		//ALARMS
	(*Input set1 L1*) 	AddError[w_Index](
			b_ErrorTrig			:= Get.Events.Input[i][phases.L1].b_alarm,
			out_ST_Error			:= a_ActiveEvents[w_Index],
			w_ErrorID					:= ((i -1) * 8) + 5,
			s_Message				:= ConcatMultiString(s1:= 'alarm: input ',
										s2:= TO_STRING(i),
			 							s3:= ' - L1: ',
										s4:= LREAL_TO_FMTSTR(Get.Events.Input[i][phases.L1].r_MaxCurrentDetected,1, TRUE),
										s5:= ' A for ',
										s6:= TO_STRING(Get.Events.Input[i][phases.L1].t_MaxTimeActive)),
			e_sev					:= eseverity.Warning,
			e_ErrAckAccess		:= eErrAckAccess.operator
			);
		w_Index := w_Index +1;
	(*Input set1 L2*) 	AddError[w_Index](
			b_ErrorTrig			:= Get.Events.Input[i][phases.L2].b_alarm,
			out_ST_Error			:= a_ActiveEvents[w_Index],
			w_ErrorID					:= ((i -1) * 8) + 6,
			s_Message				:= ConcatMultiString(s1:= 'alarm: input ',
										s2:= TO_STRING(i),
			 							s3:= ' - L2: ',
										s4:= LREAL_TO_FMTSTR(Get.Events.Input[i][phases.L2].r_MaxCurrentDetected,1, TRUE),
										s5:= ' A for ',
										s6:= TO_STRING(Get.Events.Input[i][phases.L2].t_MaxTimeActive)),
			e_sev					:= eseverity.Warning,
			e_ErrAckAccess		:= eErrAckAccess.operator
			);
		w_Index := w_Index +1;
	(*Input set1 L3*) 	AddError[w_Index](
			b_ErrorTrig			:= Get.Events.Input[i][phases.L3].b_alarm,
			out_ST_Error			:= a_ActiveEvents[w_Index],
			w_ErrorID					:= ((i -1) * 8) + 7,
			s_Message				:= ConcatMultiString(s1:= 'alarm: input ',
										s2:= TO_STRING(i),
			 							s3:= ' - L3: ',
										s4:= LREAL_TO_FMTSTR(Get.Events.Input[i][phases.L3].r_MaxCurrentDetected,1, TRUE),
										s5:= ' A for ',
										s6:= TO_STRING(Get.Events.Input[i][phases.L3].t_MaxTimeActive)),
			e_sev					:= eseverity.Warning,
			e_ErrAckAccess		:= eErrAckAccess.operator
			);
		w_Index := w_Index +1;
	(*Input set1 N*) 	AddError[w_Index](
			b_ErrorTrig			:= Get.Events.Input[i][phases.N].b_alarm,
			out_ST_Error			:= a_ActiveEvents[w_Index],
			w_ErrorID					:= ((i -1) * 8) + 8,
			s_Message				:= ConcatMultiString(s1:= 'alarm: input ',
										s2:= TO_STRING(i),
			 							s3:= ' - N: ',
										s4:= LREAL_TO_FMTSTR(Get.Events.Input[i][phases.N].r_MaxCurrentDetected,1, TRUE),
										s5:= ' A for ',
										s6:= TO_STRING(Get.Events.Input[i][phases.N].t_MaxTimeActive)),
			e_sev					:= eseverity.Warning,
			e_ErrAckAccess		:= eErrAckAccess.operator
			);
		w_Index := w_Index +1;
END_FOR

//OUTPUTS
FOR i:= 1 TO 3 DO
	//Warnings
	(*Input set1 L1*) 	AddError[w_Index](
			b_ErrorTrig			:= Get.Events.Output[i][phases.L1].b_warning,
			out_ST_Error			:= a_ActiveEvents[w_Index],
			w_ErrorID					:= ((i -1) * 8) + 17,
			s_Message				:= ConcatMultiString(s1:= 'warning: output ',
										s2:= TO_STRING(i),
			 							s3:= ' - L1: ',
										s4:= TO_STRING(Get.Events.Output[i][phases.L1].ui_actLoad),
										s5:= ' %, remaining time ',
										s6:= TO_STRING(Get.Events.Output[i][phases.L1].t_RemainingTime)),
			e_sev					:= eseverity.Warning,
			e_ErrAckAccess		:= eErrAckAccess.operator,
			b_autoClear			:= TRUE
			);
		w_Index := w_Index +1;
	(*Input set1 L2*) 	AddError[w_Index](
			b_ErrorTrig			:= Get.Events.Output[i][phases.L2].b_warning,
			out_ST_Error			:= a_ActiveEvents[w_Index],
			w_ErrorID					:= ((i -1) * 8) + 18,
			s_Message				:= ConcatMultiString(s1:= 'warning: output ',
										s2:= TO_STRING(i),
			 							s3:= ' - L2: ',
										s4:= TO_STRING(Get.Events.Output[i][phases.L2].ui_actLoad),
										s5:= ' %, remaining time ',
										s6:= TO_STRING(Get.Events.Output[i][phases.L2].t_RemainingTime)),
			e_sev					:= eseverity.Warning,
			e_ErrAckAccess		:= eErrAckAccess.operator,
			b_autoClear			:= TRUE
			);
		w_Index := w_Index +1;
	(*Input set1 L3*) 	AddError[w_Index](
			b_ErrorTrig			:= Get.Events.Output[i][phases.L3].b_warning,
			out_ST_Error			:= a_ActiveEvents[w_Index],
			w_ErrorID					:= ((i -1) * 8) + 19,
			s_Message				:= ConcatMultiString(s1:= 'warning: output ',
										s2:= TO_STRING(i),
			 							s3:= ' - L3: ',
										s4:= TO_STRING(Get.Events.Output[i][phases.L3].ui_actLoad),
										s5:= ' %, remaining time ',
										s6:= TO_STRING(Get.Events.Output[i][phases.L3].t_RemainingTime)),
			e_sev					:= eseverity.Warning,
			e_ErrAckAccess		:= eErrAckAccess.operator,
			b_autoClear			:= TRUE
			);
		w_Index := w_Index +1;
	(*Input set1 N*) 	AddError[w_Index](
			b_ErrorTrig			:= Get.Events.Output[i][phases.N].b_warning,
			out_ST_Error			:= a_ActiveEvents[w_Index],
			w_ErrorID				:= ((i -1) * 8) + 20,
			s_Message				:= ConcatMultiString(s1:= 'warning: output ',
										s2:= TO_STRING(i),
			 							s3:= ' - N: ',
										s4:= TO_STRING(Get.Events.Output[i][phases.N].ui_actLoad),
										s5:= ' %, remaining time ',
										s6:= TO_STRING(Get.Events.Output[i][phases.N].t_RemainingTime)),
			e_sev					:= eseverity.Warning,
			e_ErrAckAccess		:= eErrAckAccess.operator,
			b_autoClear			:= TRUE
			);
		w_Index := w_Index +1;
		
		//ALARMS					
	(*Output set1 L1*) 	AddError[w_Index](
			b_ErrorTrig			:= Get.Events.Output[i][phases.L1].b_alarm,
			out_ST_Error			:= a_ActiveEvents[w_Index],
			w_ErrorID					:= ((i -1) * 8) + 21,
			s_Message				:= ConcatMultiString(s1:= 'alarm: output ',
										s2:= TO_STRING(i),
			 							s3:= ' - L1: ',
										s4:= LREAL_TO_FMTSTR(Get.Events.output[i][phases.L1].r_MaxCurrentDetected,1, TRUE),
										s5:= ' A for ',
										s6:= TO_STRING(Get.Events.Output[i][phases.L1].t_MaxTimeActive)),
			e_sev					:= eseverity.Normalshutdown,
			t_triggerTime			:= st_params.OutputNormalShutdownDelay,
			e_ErrAckAccess		:= eErrAckAccess.operator
			);
		w_Index := w_Index +1;
	(*Output set1 L2*) 	AddError[w_Index](
			b_ErrorTrig			:= Get.Events.Output[i][phases.L2].b_alarm,
			out_ST_Error			:= a_ActiveEvents[w_Index],
			w_ErrorID					:= ((i -1) * 8) + 22,
			s_Message				:= ConcatMultiString(s1:= 'alarm: output ',
										s2:= TO_STRING(i),
			 							s3:= ' - L2: ',
										s4:= LREAL_TO_FMTSTR(Get.Events.output[i][phases.L2].r_MaxCurrentDetected,1, TRUE),
										s5:= ' A for ',
										s6:= TO_STRING(Get.Events.Output[i][phases.L2].t_MaxTimeActive)),
			e_sev					:= eseverity.Normalshutdown,
			t_triggerTime			:= st_params.OutputNormalShutdownDelay,
			);
		w_Index := w_Index +1;
	(*Output set1 L3*) 	AddError[w_Index](
			b_ErrorTrig			:= Get.Events.Output[i][phases.L3].b_alarm,
			out_ST_Error			:= a_ActiveEvents[w_Index],
			w_ErrorID					:= ((i -1) * 8) + 23,
			s_Message				:= ConcatMultiString(s1:= 'alarm: output ',
										s2:= TO_STRING(i),
			 							s3:= ' - L3: ',
										s4:= LREAL_TO_FMTSTR(Get.Events.output[i][phases.L3].r_MaxCurrentDetected,1, TRUE),
										s5:= ' A for ',
										s6:= TO_STRING(Get.Events.Output[i][phases.L3].t_MaxTimeActive)),
			e_sev					:= eseverity.Normalshutdown,
			t_triggerTime			:= st_params.OutputNormalShutdownDelay,
			e_ErrAckAccess		:= eErrAckAccess.operator
			);
		w_Index := w_Index +1;
	(*Output set1 N*) 	AddError[w_Index](
			b_ErrorTrig			:= Get.Events.output[i][phases.N].b_alarm,
			out_ST_Error			:= a_ActiveEvents[w_Index],
			w_ErrorID					:= ((i -1) * 8) + 24,
			s_Message				:= ConcatMultiString(s1:= 'alarm: output ',
										s2:= TO_STRING(i),
			 							s3:= ' - N: ',
										s4:= LREAL_TO_FMTSTR(Get.Events.output[i][phases.N].r_MaxCurrentDetected,1, TRUE),
										s5:= ' A for ',
										s6:= TO_STRING(Get.Events.Output[i][phases.N].t_MaxTimeActive)),
			e_sev					:= eseverity.Normalshutdown,
			t_triggerTime 			:= st_params.OutputNormalShutdownDelay,
			e_ErrAckAccess		:= eErrAckAccess.operator
			);
		w_Index := w_Index +1;
END_FOR	

(*output MCCB triggered*) 	AddError[w_Index](
			b_ErrorTrig				:= Get.b_OutputAlarm,
			out_ST_Error			:= a_ActiveEvents[w_Index],
			w_ErrorID				:= 41,
			s_Message				:= ConcatMultiString(s1:= 'Output MCCB trip. Phase: ',
										s2:= get.s_locationPeak,
			 							s3:= ', peakcurrent: ',
										s4:= LREAL_TO_FMTSTR(get.r_PeakCurrent,1, TRUE),
										s5:= ' A for ',
										s6:= TO_STRING(get.t_PeakCurrentDuration)),
			e_sev					:= eseverity.Warning
			);
		w_Index := w_Index +1;
END_METHOD

METHOD Reset : BOOL
VAR_INPUT
END_VAR

VAR_INST
	counter : INT;
END_VAR
reset := FALSE;


//reset values if it was triggered by an alarm
IF get.b_InputAlarm OR get.b_OutputAlarm OR get.r_PeakCurrent <>0 THEN
	get.r_PeakCurrent := 0;
	get.t_PeakCurrentDuration := T#0S;
	get.s_locationPeak := '';
	b_reset := TRUE;
	counter := counter +1;
ELSE
	b_reset := FALSE;
	reset := NOT b_reset;
END_IF
END_METHOD

END_FUNCTION_BLOCK

// ---- POUs/Functions-FBs-Programs/_generalFunctions/ConcatMultiString.TcPOU
FUNCTION ConcatMultiString : STRING
VAR_INPUT
	s1: STRING;
	s2: STRING;
	s3: STRING;
	s4: STRING;
	s5: STRING;
	s6: STRING;
END_VAR
VAR
END_VAR

ConcatMultiString := CONCAT(s1, CONCAT(s2, CONCAT(s3, CONCAT(s4, CONCAT(s5, s6)))));

END_FUNCTION

// ---- POUs/Objects/Enclosure/FB_Enclosure.TcPOU
FUNCTION_BLOCK FB_Enclosure
VAR_IN_OUT CONSTANT
	st_params		: ST_Enclosure_params;
END_VAR

VAR_OUTPUT
	get					: ST_Enclosure_Get;
END_VAR

VAR_INPUT
	ledstrip			: FB_ledstrip;
	set					: ST_Enclosure_set;
END_VAR

VAR
	
	climate						: FB_enclosureClimate;
	doors						: FB_DoorsNlocks;
END_VAR

ledstrip(st_params := st_params.ledstrip, get => get.ledstrip, brightness := set.by_LedBrightness);

climate( get => get.climate, st_params:= st_params.Climate);

doors(get => get.doors);

{warning 'tbd: add new enclosure door switch option'}

METHOD PUBLIC GetDiagnostics
VAR_IN_OUT
	AddError		: ARRAY [*] OF FB_AddErrorST;
	a_ActiveEvents	: ARRAY [*] OF ST_ErrorStruct;
	w_Index			: WORD;
END_VAR

VAR_OUTPUT
	b_errorActive	: BOOL;
	b_warningActive	: BOOL;
END_VAR

VAR
	by_errCt	: BYTE;
	by_warnCt	: BYTE;
END_VAR
Climate.GetDiagnostics(Adderror := AddError, a_ActiveEvents := a_ActiveEvents, w_Index := w_index);
Doors.GetDiagnostics(Adderror := AddError, a_ActiveEvents := a_ActiveEvents, w_Index := w_index);
Ledstrip.GetDiagnostics(Adderror := AddError, a_ActiveEvents := a_ActiveEvents, w_Index := w_index);
END_METHOD

METHOD GetWearCounters : BOOL
VAR_INST
	ControlCabinetDoorSwitch	:	FB_Varlogger;
	ClientPanelDoorSwitch		:	FB_Varlogger;
	
END_VAR
// ControlCabinetDoorSwitch(	TriggerInput := NOT get.doors.b_ControlPanelDoorClosed, 
// 							LogItemGroup :=  eLogItemGroupID.Enclosure, 
// 							LogItemName := 'CtrlCabDoorSwCnt', 
// 							LogType := elogtypes.TrackCycles);		
// 												
// ClientPanelDoorSwitch(	TriggerInput := NOT get.doors.b_ClientpanelDoorClosed, 
// 						LogItemGroup :=  eLogItemGroupID.Enclosure, 
// 						LogItemName := 'ClientPnlDoorSwCnt', 
// 						LogType := eLogtypes.TrackCycles);
END_METHOD

END_FUNCTION_BLOCK

// ---- POUs/Objects/Enclosure/LedIndicator/FB_Ledstrip.TcPOU
FUNCTION_BLOCK FB_Ledstrip
VAR_INPUT
	brightness						: BYTE; // in 
END_VAR

VAR_IN_OUT CONSTANT
	st_params				: st_ledstrip_params;
END_VAR

VAR_OUTPUT
	get 					: st_ledstrip_get;
END_VAR
VAR
	ledBeckhoff				: FB_ledBeckhoff;
	MachineData				: ST_Ledstrip_MachineData;
END_VAR

ledbeckhoff(Machinedata := Machinedata, st_params := st_params, Brightness := brightness, DemoMode := GVL.b_LEDDemoMode);

get := ledbeckhoff.get;

METHOD PUBLIC GetDiagnostics
VAR_IN_OUT
	AddError		: ARRAY [*] OF FB_AddErrorST;
	a_ActiveEvents	: ARRAY [*] OF ST_ErrorStruct;
	w_Index			: WORD;
END_VAR

VAR_OUTPUT
	b_errorActive	: BOOL;
	b_warningActive	: BOOL;
END_VAR

VAR
	by_errCt	: BYTE;
	by_warnCt	: BYTE;
END_VAR
	(*LED Error*)		AddError[w_Index](
		b_ErrorTrig			:= get.b_error,
		out_ST_Error			:= a_ActiveEvents[w_Index],
		w_ErrorID					:= 1,
		e_ObjectID				:=  eObject_ID.Enclosure_LED,
		s_Message				:= 'LED error',
		e_sev					:= eseverity.info,
		b_AutoClear			:= TRUE
		);
		w_Index := w_Index +1;
END_METHOD

METHOD SetMachineStatus : BOOL
VAR_INPUT
	b_Error 		: BOOL;
	b_Warning		: BOOL;
	b_Attention		: BOOL;
	b_Normal		: BOOL;
	b_Off			: BOOL;
	r_Soc			: REAL;
	r_DCcurrent		: REAL;
END_VAR

VAR_INST
	r_socDemo	: REAL := 30;
	r_CurrentDemo : REAL := 0;
END_VAR
IF b_off THEN
	machinedata.e_systemStatus := eSystemStatus.off;
ELSIF b_Error THEN
	machinedata.e_systemStatus := eSystemStatus.error;
ELSIF b_warning THEN
	machinedata.e_systemStatus := eSystemStatus.warning;
ELSIF b_attention THEN
	machinedata.e_systemStatus := eSystemStatus.attention;
ELSIF b_normal THEN
	machinedata.e_systemStatus := eSystemStatus.normal;
ELSE
	machinedata.e_systemStatus := eSystemStatus.neutral;
END_IF

MachineData.r_SOC := r_soc;
MachineData.r_DCCurrent := r_DCcurrent;
END_METHOD

END_FUNCTION_BLOCK

// ---- POUs/Objects/Enclosure/LedIndicator/BeckhoffController/FB_LedBeckhoff.TcPOU
FUNCTION_BLOCK FB_LedBeckhoff
VAR_INPUT
	Brightness				: BYTE;
	DemoMode				: BOOL;
END_VAR
VAR_OUTPUT
	get 					: st_ledstrip_get;
	Ready					: BOOL;			
END_VAR

VAR_IN_OUT CONSTANT
	MachineData				: ST_Ledstrip_machineData;
	st_params				: st_ledstrip_params;
END_VAR

VAR	
	EL2574State		AT %I* 	: UINT;
	st_LEDStatus	AT %I* 	: LEDStatus;
	st_LEDControl	AT %Q* 	: LEDControl;	
	ton_LEDdataSend		: ton := (PT:=T#300MS);
	LedsToAnimate		: BYTE		:= 5;

	ui_ActiveLeds		: UINT;
	e_LEDSteps			: eLEDSteps;
	ui_oldSOC			: UINT;
	ui_SOC 				: UINT;
	SFCStep				: UINT;
	LedBusy				: TOF := (PT := T#50MS);
	AnimationReady		: BOOL;
	
	bufferReady			: BOOL;
	ReadyToTransmit		: BOOL;
	
	GradientToggle		: BOOL;
	DemoSoc				: UINT := 50;
	DemoSocPulse		: TON := (PT:= T#500MS);
	DemoCharging		: BOOL;
END_VAR

ready := EL2574State.3;
LedBusy(IN := st_ledStatus.busy OR st_ledstatus.transmit OR st_ledstatus.error OR st_LEDControl.Execute);



IF ready THEN //AND ton_CycleTime.Q THEN
	get.BeckhoffLed := TRUE;
	
	//get system state error
	IF Machinedata.e_systemStatus = eSystemStatus.error THEN
		ui_SOC := 100;
	ELSE
		ui_SOC := REAL_TO_UINT (Machinedata.r_soc);
	END_IF
	
	//set ledstrip error to system
	get.b_Error := st_LEDStatus.error;
	
	//SOc and corresponding leds
	
	ui_ActiveLeds:= ((st_params.Numleds * ui_SOC)/100);
	
//	IF MachineData.e_systemStatus = 0 THEN
//		e_LEDSteps := eLEDSteps.initialise;
//	END_IF
	
	//setup color values and no of led according to soc. 
	CASE e_LEDSteps OF	
		eLEDSteps.initialise:
			st_LEDControl.command := 2; //Clear
			st_LEDControl.length := st_params.Numleds;
			st_LEDControl.index := 0;

			IF NOT ledbusy.Q THEN
				st_LEDControl.execute := NOT st_LEDControl.execute;
				st_LEDControl.update  := NOT st_LEDControl.update;
				e_LEDSteps := eLEDSteps.running;	
			END_IF
						

		eLEDSteps.running:	
			st_LEDControl.UPDATE 	:= FALSE;
			st_LEDControl.Execute 	:= FALSE;
			CASE SFCStep OF 
				0: 	BufferReady := FALSE;
					ReadyToTransmit := FALSE;
					st_LEDControl.command	:= 2; //Clear
					
					IF NOT LedBusy.Q THEN
						st_LEDControl.Execute 	:= NOT st_LEDControl.Execute;
						SFCStep := SEL(DemoMode, 1,2);
					END_IF
						
				1:	st_LEDControl.command	:= 1; //fill
					st_LEDControl.length 	:= ui_ActiveLeds;
					st_LEDControl.index		:= 0;
					st_LEDcontrol.parameter := 0;
					st_LEDControl.color 	:= setcolor(brightness);
					
					IF NOT LedBusy.Q THEN
						st_LEDControl.Execute 	:= NOT st_LEDControl.Execute;
						SFCStep := 3;
					END_IF
				2: //demo mode
					DemoSocPulse(IN := NOT DemoSocPulse.Q);
					IF DemoSocPulse.Q THEN
						IF DemoSoc <= 50 THEN
							DemoCharging := TRUE;
						ELSIF DemoSoc >= st_Params.Numleds THEN
							DemoCharging := FALSE;
						END_IF
						
						DemoSoc := DemoSoc + SEL(democharging, -1, 1);
					END_IF
					
					IF NOT DemoMode THEN SfcSTEP := 0; END_IF;
					st_LEDControl.length 	:= demosoc;
					st_LEDControl.index		:= 0;
					st_LEDControl.color.blue:= 0;
					
					IF NOT GradientToggle THEN
						st_LEDControl.command	:= 8; //fill
						st_LEDControl.color.Green:= 0;
						st_LEDControl.color.red:= brightness;
					ELSE
						st_LEDControl.command	:= 9; //fill
						st_LEDControl.color.Green:= brightness;
						st_LEDControl.color.red:= 0;
					END_IF
					
					IF NOT LedBusy.Q THEN
						st_LEDControl.Execute 	:= NOT st_LEDControl.Execute;
						
						IF GradientToggle THEN
							st_LEDControl.Execute := FALSE;
							SFCStep := 4;
						END_IF
						GradientToggle := NOT GradientToggle;
					END_IF
					
				3: 
					IF NOT animationReady AND NOT LedBusy.Q THEN
							AnimationReady := SetAnimation(ActiveLeds := ui_activeLeds, charging:= getChargingState() = eDCstate.charging, reset := getChargingState() = eDCstate.idle, ledstoAnimate := LedsToAnimate);
					END_IF
					
					IF AnimationReady THEN
						AnimationReady := FALSE;
						st_LEDControl.Execute := NOT st_LEDControl.Execute;
						SFCStep := SFCStep + 1;
					END_IF
				ELSE
					bufferReady := TRUE;
			END_CASE
			
			ton_LEDdataSend(in:= NOT ton_LEDdataSend.Q AND bufferReady);
			IF ton_LEDDataSend.Q THEN
				ReadyToTransmit := TRUE;
			END_IF
			
			IF ReadyToTransmit AND NOT ledbusy.Q THEN
				SFCStep := 0;
				st_LEDControl.UPDATE 	:= NOT st_LEDControl.UPDATE;
				st_LEDControl.Execute 	:= NOT st_LEDControl.execute;	
			END_IF		
	END_CASE
END_IF

METHOD GetChargingState : eDCstate; 
VAR_INPUT
END_VAR
IF machinedata.r_DCCurrent > 10 THEN
	GetChargingState := eDCstate.discharging;
	//b_charging := FALSE;	
	//b_discharging := TRUE;
ELSIF machinedata.r_DCCurrent < -10 THEN
	GetChargingState := eDCstate.charging;
	//b_charging := TRUE;
	//b_discharging := FALSE;
ELSE
	GetChargingState := eDCstate.idle;
	//b_discharging := FALSE;
	//b_charging := FALSE;	
END_IF
END_METHOD

METHOD SetAnimation : BOOL;
VAR_INPUT
	ActiveLeds			: UINT;
	Charging			: BOOL;
	reset				: BOOL;
	LedsToAnimate		: BYTE := 5;	
END_VAR

VAR_INST
	AnimateResetToggle	: BYTE;
	//moveCounter			: CTUD;
	//ready				: BOOL;
	ledcounter			: BYTE;
END_VAR

//movecounter(pv := LedsToAnimate +1);
//moveCounter.LOAD := moveCounter.QD AND Charging;
//moveCounter.Reset := moveCounter.CV > movecounter.PV AND NOT Charging OR Reset;

//CASE AnimateResetToggle OF
//0:		AnimateResetToggle := AnimateResetToggle +1;
//		moveCounter.CU := FALSE;
//		moveCounter.CD := FALSE;
//	ELSE
//		AnimateResetToggle := 0;
//		moveCounter.cu := NOT charging;
//		movecounter.cd := Charging;
//		st_LEDControl.length 	:= 1;
//		st_LEDControl.command	:= 1; //move
//		st_LEDControl.parameter := 0;
//		st_LEDControl.index :=  ui_ActiveLeds + moveCounter.CV -1;
//		SetAnimation := TRUE;
//END_CASE

IF NOT RESET THEN
	ledcounter := ledcounter + SEL(charging,1 ,-1);
	IF ledcounter >= LedsToAnimate * 2 OR ledcounter = 0 THEN
		ledcounter := SEL(charging,0 ,LedsToAnimate * 2);	 
	END_IF
	
	st_LEDControl.length 	:= 1;
	st_LEDControl.command	:= 1; //move
	st_LEDControl.parameter := 
	st_LEDControl.index :=  ActiveLeds + ledcounter/2;
ELSE
	ledcounter := 0;
END_IF

SetAnimation := TRUE;
END_METHOD

METHOD SetColor : LEDColor

VAR_INPUT
	Brightness		: BYTE;
END_VAR

VAR
	tempColorValue	: USINT;
END_VAR
CASE machinedata.e_systemStatus OF
	eSystemStatus.neutral: 		
		SetColor.blue	:= Brightness;
		SetColor.red	:= Brightness;
		SetColor.green	:= Brightness;

	eSystemStatus.normal: 
		SetColor.blue	:= 0;
		SetColor.red	:= 0;
		SetColor.green	:= Brightness;
	
	eSystemStatus.attention: 
		SetColor.blue	:= Brightness;
		SetColor.red	:= 0;
		SetColor.green	:= 0;
	eSystemStatus.warning: //yelow
		SetColor.blue	:= 0;
		SetColor.red	:= Brightness;
		SetColor.green	:= Brightness/3;
	
	eSystemStatus.error: 
		SetColor.blue	:= 0;
		SetColor.red	:= Brightness;
		SetColor.green	:= 0;	
END_CASE

//Change RGB order
IF st_params.ColorOrder = eColorOrder.GRB THEN
	tempColorValue := setColor.Red;
	setcolor.red := setcolor.green;
	SetColor.green := tempColorValue;
END_IF
END_METHOD

END_FUNCTION_BLOCK

// ---- POUs/Objects/Enclosure/Climate/FB_EnclosureClimate.TcPOU
FUNCTION_BLOCK FB_EnclosureClimate
VAR_IN_OUT CONSTANT
	st_params				: ST_EnclosureClimate_params;
END_VAR
VAR_OUTPUT
	get						: ST_EnclosureClimate_get;
END_VAR

VAR
	TempRead		AT %I* : ST_AnalogInputData;
	HumRead			AT %I* : ST_AnalogInputData;
	
	scaleTemp				: FB_CTRL_SCALE;
	scaleHum				: FB_CTRL_SCALE;
	scaleParams				: ST_CTRL_SCALE_Params;
END_VAR

scaleParams.tCtrlCycleTime := T#100MS;
	scaleParams.tTaskCycleTime := T#1MS;
	scaleParams.fInMax := 16#7FFF;
	scaleParams.fInMin := 16#0000;
	scaleParams.fOutMax := 60;
	scaleParams.fOutMin:= -40;

scaleTemp(fin := TempRead.Value, fout => get.r_Temperature, stParams := scaleParams);
scaleParams.fOutMax := 100;
scaleParams.fOutMin := 0;
scaleHum(fin := HumRead.Value, fout => get.r_Humidity, stParams := scaleParams);

CalculateDewpoint();

METHOD CalculateDewpoint : REAL;
var
	Alpha : real;
END_VAR
alpha := LN(MAX(get.r_Humidity,0.01)/100)+(17.625*get.r_Temperature/(243.12+get.r_Temperature));
get.r_Dewpoint := 243.12*alpha/(17.625-alpha);
END_METHOD

METHOD EnclosureConditioning : eConditioningRequirement;
VAR_INST
	HeatingRequired : SR;
	CoolingRequired : SR;
END_VAR

VAR_INPUT
	b_Reset	:	BOOL := FALSE;
END_VAR
	
// TODO: test 123

HeatingRequired.SET := get.r_Temperature < MAX(st_params.r_EnclosureConditioningTempMin, get.r_Dewpoint);
HeatingRequired.Reset := get.r_Temperature > MAX(st_params.r_EnclosureConditioningTempMin, r_Enclosuredewpoint) + st_params.r_TemperatureHysteris OR b_Reset;

CoolingRequired.SET := get.r_Temperature > st_params.r_EnclosureIdleTempMax;
CoolingRequired.Reset := get.r_Temperature < MAX(st_params.r_EnclosureIdleTempMax-5) OR b_Reset;

IF CoolingRequired.Q1 THEN
	EnclosureConditioning := eConditioningRequirement.CoolingRequired;
ELSIF HeatingRequired.Q1 THEN
	EnclosureConditioning := eConditioningRequirement.HeatingRequired;
ELSE
	EnclosureConditioning := eConditioningRequirement.none;
END_IF
END_METHOD

METHOD PUBLIC GetDiagnostics
VAR_IN_OUT
	AddError		: ARRAY [*] OF FB_AddErrorST;
	a_ActiveEvents	: ARRAY [*] OF ST_ErrorStruct;
	w_Index			: WORD;
END_VAR


VAR
	by_errCt	: BYTE;
	by_warnCt	: BYTE;
END_VAR
	(*Humidity High*)		AddError[w_Index](
		b_ErrorTrig			:= get.events.b_HumidityHigh,
		out_ST_Error			:= a_ActiveEvents[w_Index],
		w_ErrorID					:= 1,
		e_ObjectID				:=  eObject_ID.Enclosure_climate,
		s_Message				:= 'humidity high',
		e_sev					:= eseverity.Warning,
		b_AutoClear			:= TRUE
		);
		w_Index := w_Index +1;
	
	(*Humidity Too High*)		AddError[w_Index](
		b_ErrorTrig			:= get.events.b_HumidityTooHigh,
		out_ST_Error			:= a_ActiveEvents[w_Index],
		w_ErrorID					:= 2,
		s_Message				:= 'humidity too high',
		e_sev					:= eseverity.QuickShutdown,
		e_ErrAckAccess		:= eErrAckAccess.Operator
	);
	w_Index := w_Index +1;
	
	(*Temperature High*)		AddError[w_Index](
		b_ErrorTrig			:= get.events.b_TemperatureHigh,
		out_ST_Error			:= a_ActiveEvents[w_Index],
		w_ErrorID					:= 3,
		s_Message				:= 'temperature high',
		e_sev					:= eseverity.warning,
		b_AutoClear			:= TRUE
	);
	w_Index := w_Index +1;
	
	(*Temperature Too High*)	AddError[w_Index](
		b_ErrorTrig			:= get.events.b_TemperatureTooHigh,
		out_ST_Error			:= a_ActiveEvents[w_Index],
		w_ErrorID					:= 4,
		s_Message				:= 'temperature too high',
		e_sev					:= eseverity.Quickshutdown,
		e_ErrAckAccess		:= eErrAckAccess.Operator
	);

	w_Index := w_Index +1;
	
	(*Temperature Low*)	AddError[w_Index](
		b_ErrorTrig			:= get.events.b_TemperatureLow,
		out_ST_Error			:= a_ActiveEvents[w_Index],
		w_ErrorID					:= 5,
		s_Message				:= 'temperature low',
		e_sev					:= eseverity.Warning,
		b_AutoClear			:= TRUE
	);
	w_Index := w_Index +1;
	
	(*Temperature Too Low*)	AddError[w_Index](
		b_ErrorTrig			:= get.events.b_TemperatureTooLow,
		out_ST_Error			:= a_ActiveEvents[w_Index],
		w_ErrorID					:= 6,
		s_Message				:= 'temperature too low',
		e_sev					:= eseverity.Normalshutdown,
		e_ErrAckAccess		:= eErrAckAccess.Operator
	);
	w_Index := w_Index +1;
	
	(*4-20ma Overrange*)	AddError[w_Index](
		b_ErrorTrig			:= get.events.b_AIOverrange,
		out_ST_Error			:= a_ActiveEvents[w_Index],
		w_ErrorID					:= 7,
		s_Message				:= 'analog input temp/humid overrange',
		e_sev					:= eseverity.Warning,
		b_AutoClear			:= TRUE
	);
	w_Index := w_Index +1;
	
	(*4-20ma Underrange*)	AddError[w_Index](
		b_ErrorTrig			:= get.events.b_AIUnderrange,
		out_ST_Error			:= a_ActiveEvents[w_Index],
		w_ErrorID					:= 8,
		s_Message				:= 'analog input temp/humid underrange',
		e_sev					:= eseverity.Warning,
		b_AutoClear			:= TRUE
	);
	w_Index := w_Index +1;
	
	(*Analog input error*)	AddError[w_Index](
		b_ErrorTrig			:= get.events.b_AIError,
		out_ST_Error			:= a_ActiveEvents[w_Index],
		w_ErrorID					:= 9,
		s_Message				:= 'analog input temp/humid error',
		e_sev					:= eseverity.warning,
		b_AutoClear			:= TRUE
	);
	w_Index := w_Index +1;
	
	(*Analog input error*)	AddError[w_Index](
		b_ErrorTrig				:= get.events.b_DewpointTooHigh,
		out_ST_Error			:= a_ActiveEvents[w_Index],
		w_ErrorID				:= 10,
		s_Message				:= 'dewpoint too high alarm',
		e_sev					:= eseverity.normalshutdown,
	);
	w_Index := w_Index +1;
END_METHOD

METHOD PRIVATE SetEvents : BOOL
VAR_IN_OUT
	get : ST_EnclosureClimate_get;
	st_params : ST_EnclosureClimate_params;
END_VAR

VAR_INST
	sr_HumHigh			: SR;
	sr_HumTooHigh		: SR;
	sr_TempHigh			: SR;
	sr_TempTooHigh		: SR;
	sr_TempLow			: SR;
	sr_TempTooLow		: SR;
END_VAR
//set events
get.events.b_AIError := TempRead.Status.Error OR HumRead.Status.Error;
get.events.b_AIUnderrange := TempRead.Status.Underrange OR HumRead.Status.Underrange;
get.events.b_AIOverrange := TempRead.Status.Overrange OR HumRead.Status.Overrange;

sr_HumHigh(
	SET1:= get.r_Humidity > st_params.r_HumidityHigh, 
	RESET:= get.r_Humidity <= st_params.r_HumidityHigh - st_params.r_HumidityHysteris,
	Q1 => get.events.b_HumidityHigh);
sr_HumTooHigh(
	SET1:= get.r_Humidity > st_params.r_HumidityTooHigh, 
	RESET:= get.r_Humidity <= st_params.r_HumidityTooHigh - st_params.r_HumidityHysteris,
	Q1 => get.events.b_HumidityTooHigh);	
sr_TempHigh(
	SET1:= get.r_Temperature > st_params.r_TemperatureHigh, 
	RESET:= get.r_Temperature <= st_params.r_TemperatureHigh - st_params.r_TemperatureHysteris,
	Q1 => get.events.b_TemperatureHigh);	
sr_TempTooHigh(
	SET1:= get.r_Temperature > st_params.r_TemperatureTooHigh, 
	RESET:= get.r_Temperature <= st_params.r_TemperatureTooHigh - st_params.r_TemperatureHysteris,
	Q1 => get.events.b_TemperatureTooHigh);
sr_TempLow(
	SET1:= get.r_Temperature < st_params.r_TemperatureLow, 
	RESET:= get.r_Temperature >= st_params.r_TemperatureLow + st_params.r_TemperatureHysteris,
	Q1 => get.events.b_TemperatureLow);
sr_TempTooLow(
	SET1:= get.r_Temperature < st_params.r_TemperatureTooLow, 
	RESET:= get.r_Temperature >= st_params.r_TemperatureTooLow + st_params.r_TemperatureHysteris,
	Q1 => get.events.b_TemperatureTooLow);
END_METHOD

END_FUNCTION_BLOCK

// ---- POUs/Objects/Enclosure/Doors/FB_DoorsNLocks.TcPOU
FUNCTION_BLOCK FB_DoorsNLocks
VAR_OUTPUT
	get 		: ST_DoorsNLocks_get;
END_VAR

VAR_INPUT
	b_DoorswitchOptionFitted	: BOOL;
END_VAR

VAR
	b_ControlPanelDoorfb		AT %I* : BOOL;
	b_ClientPanelDoorfb			AT %I* : BOOL;
	b_InverterDoorOpen			AT %I* : BOOL;
	b_UPSBatteryDoorOpen		AT %I* : BOOL;
    b_MainBatteryLeftDoorOpen	AT %I* : BOOL;
    b_MainBatteryRightDoorOpen	AT %I* : BOOL;
	BusCouplerState				AT %I* : UINT;
END_VAR


if b_DoorswitchOptionFitted then
	get.b_BuscouplerOK := BusCouplerState = 8;
	
	get.b_ControlPanelDoorOpen 		:= get.b_BuscouplerOK and not b_ControlPanelDoorfb;
	get.b_ClientPanelDoorOpen		:= get.b_BuscouplerOK and not b_ClientPanelDoorfb; 
	get.b_InverterDoorOpen			:= get.b_BuscouplerOK and not b_InverterDoorOpen;	     
	get.b_UPSBatteryDoorOpen		:= get.b_BuscouplerOK and not b_UPSBatteryDoorOpen;		    
	get.b_MainBatteryLeftDoorOpen	:= get.b_BuscouplerOK and not b_MainBatteryLeftDoorOpen;	
	get.b_MainBatteryRightDoorOpen  := get.b_BuscouplerOK and not b_MainBatteryRightDoorOpen;
else
	get.b_ControlPanelDoorOpen 		:= false;
    get.b_ClientPanelDoorOpen		:= false;
    get.b_InverterDoorOpen			:= false;
    get.b_UPSBatteryDoorOpen		:= false;
    get.b_MainBatteryLeftDoorOpen	:= false;
    get.b_MainBatteryRightDoorOpen  := false;
END_IF

METHOD PUBLIC GetDiagnostics
VAR_IN_OUT
	AddError		: ARRAY [*] OF FB_AddErrorST;
	a_ActiveEvents	: ARRAY [*] OF ST_ErrorStruct;
	w_Index			: WORD;
END_VAR

VAR_OUTPUT
	b_errorActive	: BOOL;
	b_warningActive	: BOOL;
END_VAR

VAR
	by_errCt	: BYTE;
	by_warnCt	: BYTE;
END_VAR
AddError[w_Index](
		b_ErrorTrig				:= get.b_ClientpanelDoorOpen,
		out_ST_Error			:= a_ActiveEvents[w_Index],
		w_ErrorID				:= 1,
		e_ObjectID				:=  eObject_ID.Enclosure_doors,
		s_Message				:= 'clientpanel door opened',
		e_sev					:= eseverity.info,
		b_AutoClear				:= TRUE
		);
		w_Index := w_Index +1;
		
AddError[w_Index](
		b_ErrorTrig				:= get.b_ControlPanelDoorOpen,
		out_ST_Error			:= a_ActiveEvents[w_Index],
		w_ErrorID				:= 2,
		s_Message				:= 'controlpanel door opened',
		e_sev					:= eseverity.info,
		b_AutoClear				:= TRUE,
		);
		w_Index := w_Index +1;
		
AddError[w_Index](
		b_ErrorTrig				:= get.b_InverterDoorOpen,
		out_ST_Error			:= a_ActiveEvents[w_Index],
		w_ErrorID				:= 3,
		s_Message				:= 'Inverter door opened',
		e_sev					:= eseverity.info,
		b_AutoClear				:= TRUE
		);
		w_Index := w_Index +1;
		
AddError[w_Index](
		b_ErrorTrig				:= get.b_MainBatteryLeftDoorOpen,
		out_ST_Error			:= a_ActiveEvents[w_Index],
		w_ErrorID				:= 4,
		s_Message				:= 'Left main battery door opened',
		e_sev					:= eseverity.info,
		b_AutoClear				:= TRUE
		);
		w_Index := w_Index +1;
		
AddError[w_Index](
		b_ErrorTrig				:= get.b_MainBatteryRightDoorOpen,
		out_ST_Error			:= a_ActiveEvents[w_Index],
		w_ErrorID				:= 5,
		s_Message				:= 'Right main battery door opened',
		e_sev					:= eseverity.info,
		b_AutoClear				:= TRUE
		);
		w_Index := w_Index +1;

AddError[w_Index](
		b_ErrorTrig				:= get.b_UPSBatteryDoorOpen,
		out_ST_Error			:= a_ActiveEvents[w_Index],
		w_ErrorID				:= 6,
		s_Message				:= 'UPS battery door opened',
		e_sev					:= eseverity.info,
		b_AutoClear				:= TRUE
		);
		w_Index := w_Index +1;
		
AddError[w_Index](
		b_ErrorTrig				:= b_DoorswitchOptionFitted and not get.b_BuscouplerOK,
		out_ST_Error			:= a_ActiveEvents[w_Index],
		w_ErrorID				:= 7,
		s_Message				:= 'Doorswitch IO module inoperative',
		e_sev					:= eseverity.info,
		b_AutoClear				:= TRUE
		);
		w_Index := w_Index +1;
END_METHOD

END_FUNCTION_BLOCK

// ---- POUs/Objects/PLCStatus/FB_PLCState.TcPOU
FUNCTION_BLOCK FB_PLCState
VAR_OUTPUT
	EL9410					AT %I* : ST_EL9410;
	get							: ST_PLCstate_get;
END_VAR
VAR
	ton_refreshpulse					: TON := (PT := T#500ms);
	events : ST_PLC_events;
	by_PNErrorsAllowed					: BYTE;
	ui_EthercatMasterState		AT %I* : UINT;
	ui_ProfinetNoErrorDevices	AT %I* : UINT;
	ui_ProfinetNoDiagDevices	AT %I* : UINT;
	ui_SafetyLogicState			AT %I* : UINT;	
	
	ton_SystemReady					: TON := (IN := FALSE, PT := T#15S);	
	
	fb_cpuload 						: TC_CpuUsage;
	
END_VAR

events.b_EthercatMasterFault := ui_EthercatMasterState <> 0;

ton_SystemReady(IN:= TRUE);
GVL.b_SystemReady	:= ton_SystemReady.Q;

IF settings.Configuration.e_PNcouplerType = 0 THEN
	by_PNErrorsAllowed := 3;
ELSE 
	by_PNErrorsAllowed := 2;
END_IF

// get cpu load
ton_refreshpulse(IN := NOT ton_refreshpulse.Q);
fb_cpuload(start:= ton_refreshpulse.Q,
	TMOUT:= T#5S);
get.r_CPUload:= TO_REAL(fb_cpuload.USAGE);

IF ui_ProfinetNoErrorDevices > by_PNErrorsAllowed THEN
	get.e_ProfinetState := eNetcomState.Error;
ELSIF ui_ProfinetNoDiagDevices > by_PNErrorsAllowed THEN
	get.e_ProfinetState := eNetcomState.Warning;
ELSIF ui_ProfinetNoErrorDevices <= by_PNErrorsAllowed AND ui_ProfinetNoDiagDevices <= by_PNErrorsAllowed THEN
	get.e_ProfinetState := eNetcomState.OK;
ELSE
	get.e_ProfinetState := eNetcomState.NotConnected;
END_IF

IF ui_EthercatMasterState = 0 THEN
	get.e_EthercatState := eNetcomState.OK;
ELSIF ui_EthercatMasterState = 1 THEN
	get.e_EthercatState := eNetcomState.NotConnected;
ELSE
	get.e_EthercatState := eNetcomState.Error;
END_IF

METHOD GetDiagnostics
VAR_IN_OUT
	AddError		: ARRAY [*] OF FB_AddErrorST;
	a_ActiveEvents	: ARRAY [*] OF ST_ErrorStruct;
	w_Index			: WORD;
END_VAR
(*PLC io supply fault*)		AddError[w_Index](
					b_ErrorTrig			:= EL9410.bit_UpUndervoltage OR EL9410.bit_UsUndervoltage,
					out_ST_Error			:= a_ActiveEvents[w_Index],
					w_ErrorID					:= 1,
					e_ObjectID				:= eObject_ID.PLC,
					s_Message				:= 'EL9410 supply fault',
					e_sev					:= eSeverity.Quickshutdown
				);
				w_Index := w_Index +1;
				
(*Ethercat master fault*)		AddError[w_Index](
					b_ErrorTrig			:= events.b_EthercatMasterFault,
					out_ST_Error			:= a_ActiveEvents[w_Index],
					w_ErrorID					:= 2,
					s_Message				:= 'Ethercat master fault',
					e_sev					:= eSeverity.normalshutdown,
				);
				w_Index := w_Index +1;
END_METHOD

END_FUNCTION_BLOCK

// ---- POUs/Objects/PeakshaveBox/FB_PeakshaveBox.TcPOU
FUNCTION_BLOCK FB_PeakshaveBox
VAR_IN_OUT CONSTANT
	st_params 			: ST_peakshavebox_params;
END_VAR

VAR_INPUT
	set					: ST_peakshaveBox_set;
END_VAR

VAR_OUTPUT
	get					: ST_PeakshaveBox_get; 
END_VAR

VAR
	EmptyGet				: ST_PeakshaveBox_get;
	Buscoupler				: FB_EK1100;
	Powermeter				: FB_EL3453;

	ton_activationDelay		: TON := (PT := T#2S);
END_VAR

VAR_INPUT
	b_enable			: BOOL;
END_VAR

VAR PERSISTENT
	setpersist 					: ST_PeakshaveBox_set;
END_VAR

ton_activationDelay(IN := get.b_dataOK AND b_enable AND get.b_buscouplerReady, Q => get.b_active);// AND NOT Powermonitor.get.StatusWord.b_Error;
//Instantiate FBs

//PSB settings can only be updated when not active
IF NOT b_enable THEN
	setpersist := set;
END_IF

get.b_SettingsChangePending := MEMCMP(ADR(set), ADR(setpersist), SIZEOF(set)) <> 0;
 

Buscoupler();
Powermeter(Quality => get.PowerQuality);
Datamapping(set:=setPersist, data := get.Powermonitor);	

IF get.b_active THEN
	get.PSBmode := ePSBMode.Monitor;
	IF setpersist.b_BreakerControl THEN
		get.PSBmode := ePSBMode.MonitorControl;
	END_IF
ELSE
	get.PSBmode := ePSBMode.None;
END_IF

METHOD PUBLIC GetDiagnostics
VAR_IN_OUT
	AddError		: ARRAY [*] OF FB_AddErrorST;
	a_ActiveEvents	: ARRAY [*] OF ST_ErrorStruct;
	w_Index			: WORD;
END_VAR
(*Voltage L1 fault*) 	AddError[w_Index](
			b_ErrorTrig			:= NOT Get.b_buscouplerReady AND b_enable,
			out_ST_Error			:= a_ActiveEvents[w_Index],
			w_ErrorID				:= 1,
			e_ObjectID				:= eObject_ID.PeakshaveBox,
			s_Message				:= 'Buscoupler not detected',
			e_sev					:= eseverity.Warning,
			b_autoClear				:= TRUE
			);
		w_Index := w_Index +1;


(*Voltage L1 fault*) 	AddError[w_Index](
			b_ErrorTrig			:= Get.Powerstatus.b_Error_Phase[1],
			out_ST_Error			:= a_ActiveEvents[w_Index],
			w_ErrorID				:= 2,
			e_ObjectID				:= eObject_ID.PeakshaveBox,
			s_Message				:= 'L1 error',
			e_sev					:= eseverity.Warning,
			b_autoClear				:= TRUE
			);
		w_Index := w_Index +1;
		
(*Voltage L2 fault*) 	AddError[w_Index](
			b_ErrorTrig			:= Get.Powerstatus.b_Error_Phase[2],
			out_ST_Error			:= a_ActiveEvents[w_Index],
			w_ErrorID				:= 3,
			e_ObjectID				:= eObject_ID.PeakshaveBox,
			s_Message				:= 'L2 error',
			e_sev					:= eseverity.Warning,
			b_autoClear				:= TRUE
			);
		w_Index := w_Index +1;
		
(*Voltage L3 fault*) 	AddError[w_Index](
			b_ErrorTrig			:= Get.Powerstatus.b_Error_Phase[3],
			out_ST_Error			:= a_ActiveEvents[w_Index],
			w_ErrorID				:= 4,
			e_ObjectID				:= eObject_ID.PeakshaveBox,
			s_Message				:= 'L3 error',
			e_sev					:= eseverity.Warning,
			b_autoClear				:= TRUE
			);
		w_Index := w_Index +1;
		
(*Powermonitor current L1 out of range*) 	AddError[w_Index](
			b_ErrorTrig			:= Get.PowerStatus.b_OverCurrent AND Get.PowerStatus.b_Error_Phase[1],
			out_ST_Error			:= a_ActiveEvents[w_Index],
			w_ErrorID				:= 6,
			e_ObjectID				:= eObject_ID.PeakshaveBox,
			s_Message				:= 'Powermonitor current L1 out of range',
			e_sev					:= eseverity.Warning,
			b_autoClear				:= TRUE
			);
		w_Index := w_Index +1;
		
(*Powermonitor current L2 out of range*) 	AddError[w_Index](
			b_ErrorTrig			:= Get.PowerStatus.b_OverCurrent AND Get.PowerStatus.b_Error_Phase[2],
			out_ST_Error			:= a_ActiveEvents[w_Index],
			w_ErrorID				:= 7,
			e_ObjectID				:= eObject_ID.PeakshaveBox,
			s_Message				:= 'Powermonitor current L2 out of range',
			e_sev					:= eseverity.Warning,
			b_autoClear				:= TRUE
			);
		w_Index := w_Index +1;
		
(*Powermonitor current L3 out of range*) 	AddError[w_Index](
			b_ErrorTrig			:= Get.PowerStatus.b_OverCurrent AND Get.PowerStatus.b_Error_Phase[3],
			out_ST_Error			:= a_ActiveEvents[w_Index],
			w_ErrorID				:= 8,
			e_ObjectID				:= eObject_ID.PeakshaveBox,
			s_Message				:= 'Powermonitor current L3 out of range',
			e_sev					:= eseverity.Warning,
			b_autoClear				:= TRUE
			);
		w_Index := w_Index +1;

(*Powermonitor overcurrent fault*) 	AddError[w_Index](
			b_ErrorTrig				:= Get.PowerStatus.b_OverCurrent,
			out_ST_Error			:= a_ActiveEvents[w_Index],
			w_ErrorID				:= 11,
			e_ObjectID				:= eObject_ID.PeakshaveBox,
			s_Message				:= 'Powermonitor overcurrent fault',
			e_sev					:= eseverity.Warning,
			b_autoClear				:= TRUE
			);
		w_Index := w_Index +1;
		
(*Powermonitor overvoltage fault*) 	AddError[w_Index](
			b_ErrorTrig				:= Get.PowerStatus.b_OverVoltage,
			out_ST_Error			:= a_ActiveEvents[w_Index],
			w_ErrorID				:= 12,
			e_ObjectID				:= eObject_ID.PeakshaveBox,
			s_Message				:= 'Powermonitor overvoltage fault',
			e_sev					:= eseverity.Warning,
			b_autoClear				:= TRUE
			);
		w_Index := w_Index +1;
		
(*Powermonitor undervoltage fault*) 	AddError[w_Index](
			b_ErrorTrig				:= Get.PowerStatus.b_UnderVoltage,
			out_ST_Error			:= a_ActiveEvents[w_Index],
			w_ErrorID				:= 13,
			e_ObjectID				:= eObject_ID.PeakshaveBox,
			s_Message				:= 'Powermonitor undervoltage fault',
			e_sev					:= eseverity.Warning,
			b_autoClear				:= TRUE
			);
		w_Index := w_Index +1;

	
	(*Setting change pending*) 	AddError[w_Index](
			b_ErrorTrig				:= get.b_SettingsChangePending,
			out_ST_Error			:= a_ActiveEvents[w_Index],
			w_ErrorID				:= 14,
			e_ObjectID				:= eObject_ID.PeakshaveBox,
			s_Message				:= 'PSB settings change blocked, disable PSB to apply',
			e_sev					:= eseverity.Warning,
			b_autoClear				:= TRUE
			);
		w_Index := w_Index +1;
END_METHOD

METHOD Datamapping : BOOL

VAR_IN_OUT
	set : ST_PeakshaveBox_set; 
	data : st_PQVoltageData;
END_VAR

VAR
	i : INT;
END_VAR

VAR_INST
	FrequencyOKLowLimit  : REAL := 45;
	FrequencyOKHighLimit : REAL := 65;
	OverCurrentThreshold : REAL := 1.05;

	PhaseError: BOOL;
END_VAR
get.b_buscouplerReady := Buscoupler.state = 8 AND Powermeter.Diagnostics.State = 8;

IF NOT get.b_buscouplerReady THEN
	get := EmptyGet;	
ELSE
	Powermeter.DynamicRatio(Vprimair:= set.r_VtPrimair, VSecundair := set.r_VtSecundair, CtRatio := set.ui_CtRange, CTInverse := set.b_InverseCTdirection,
	Status => get.PowerStatus,
	ar_phaseVoltage => data.ar_PhaseVoltage,
	ar_lineVoltage	=> data.ar_LineVoltage,
	ar_Current		=> data.ar_Current,
	ar_ActivePower	=> data.ar_ActivePower,
	ar_reactivePower => data.ar_ReactivePower,
	ar_ApparentPower => data.ar_ApparentPower,
	ar_PowerFactor	=> data.ar_PowerFactor,
	ar_Frequency	=> data.ar_Frequency,
	r_VoltageUnbalance => data.r_VoltageUnbalance,
	r_CurrentUnbalance => data.r_CurrentUnbalance,
	b_VoltagesOK => data.b_VoltagesOK,
	e_ACRotationState => data.e_ACrotationStatus
);
	
END_IF
END_METHOD

END_FUNCTION_BLOCK

// ---- POUs/Functions-FBs-Programs/IO_modules/Beckhoff/FB_EK1100.TcPOU
FUNCTION_BLOCK FB_EK1100
VAR_OUTPUT
	state						AT %I* : UINT;
END_VAR

END_FUNCTION_BLOCK

// ---- POUs/Objects/GenComm/FB_GenComm.TcPOU
FUNCTION_BLOCK FB_GenComm
VAR_INPUT
	Set				:	ST_Genset_Set;
END_VAR
VAR_OUTPUT
	Get				:	ST_Genset_Get;
END_VAR
VAR
	GenCommEnable		:	BOOL 	:= TRUE;
	OverwriteSetStruct	: 	BOOL 	:= FALSE;
	AGC150 				: 	FB_AGC150;
END_VAR

VAR_IN_OUT CONSTANT
	st_params 			: ST_GenComm_params;
END_VAR

AGC150(get := get, enable := GenCommEnable AND set.enable);

IF NOT OverwriteSetStruct THEN
	CASE st_params.GenControlProtocol OF
		eGenControlProtocol.AGC150:
			AGC150.set.ip := st_params.IP;
			AGC150.set.AutoStartStop := set.StartStop;
			AGC150.set.DroopEnable := FALSE;
			//defaults:
			AGC150.set.VoltRegulator := 0;
			AGC150.set.FreqRegulator := 0;
			AGC150.set.Pset := 0;
			AGC150.set.Qset := 0;
			AGC150.set.PFset := 1;	
			CASE set.GensetMode OF
				eGensetMode.Droop:
					AGC150.set.DroopEnable := TRUE;
					//AGC150.set.MainBreakerON := eOnOffState.Disable;
					AGC150.set.U_FDroopSet := set.U_FDroopSet;
					AGC150.set.VoltRegulator := set.Uset;
					AGC150.set.FreqRegulator := set.Fset;
					AGC150.set.bIslandModeEnable := TRUE; 
					AGC150.set.bFixedPowerEnable := FALSE;
				eGensetMode.Isochronous:
					AGC150.set.DroopEnable := FALSE;
					//AGC150.set.MainBreakerON := eOnOffState.Disable;
					AGC150.set.VoltRegulator := set.Uset;
					AGC150.set.FreqRegulator := set.Fset;
					AGC150.set.bIslandModeEnable := TRUE; 
					AGC150.set.bFixedPowerEnable := FALSE;
				eGensetMode.FixedPower:
					AGC150.set.bIslandModeEnable := FALSE; 
					AGC150.set.bFixedPowerEnable := TRUE;
					AGC150.set.DroopEnable := FALSE;
					//AGC150.set.MainBreakerON := eOnOffState.enable;
					AGC150.set.Pset := set.Pset;
					AGC150.set.Qset := set.Qset;
					AGC150.set.PFset := set.PFset;
			END_CASE
	END_CASE
END_IF

METHOD GetDiagnostics
VAR_IN_OUT
	AddError		: ARRAY [*] OF FB_AddErrorST;
	a_ActiveEvents	: ARRAY [*] OF ST_ErrorStruct;
	w_Index			: WORD;
END_VAR
	(*Comm error*)		AddError[w_Index](
					b_ErrorTrig				:= NOT get.CommunicationOK AND set.enable AND st_params.GenControlProtocol <> 0,
					out_ST_Error			:= a_ActiveEvents[w_Index],
					w_ErrorID				:= 1,
					e_ObjectID				:= eObject_ID.Genset,
					s_Message				:= 'communication not ok',
					e_sev					:= eSeverity.Info
				);
				w_Index := w_Index +1;
	
		(*Fuel low*)		AddError[w_Index](
					b_ErrorTrig				:= get.FuelLow OR get.FuelCritical,
					out_ST_Error			:= a_ActiveEvents[w_Index],
					w_ErrorID				:= 2,
					e_ObjectID				:= eObject_ID.Genset,
					s_Message				:= SEL(get.FuelCritical,'fuel at low level','fuel at critically low level'),
					e_sev					:= eSeverity.Info
				);
				w_Index := w_Index +1;
END_METHOD

END_FUNCTION_BLOCK

// ---- POUs/Objects/GenComm/FB_AGC150.TcPOU
FUNCTION_BLOCK FB_AGC150

VAR_IN_OUT
	get				: ST_GENSET_Get;
END_VAR

VAR_INPUT
	enable 	: BOOL;
	set 	: ST_AGC150_set;
END_VAR

VAR
	b_changeEndianess	:	BOOL	:=	FALSE;
	ComOKRelease		:   TON := (PT:= T#5S);
	MBWriteCoils		:	FB_MBWriteCoils;	// function 15
	CoilData			:	ARRAY[0..10] OF BYTE;
	StartCoilWrite		:	BOOL;
	
	MBWriteHolding		:	FB_MBWriteRegs;		// function 16
	HoldingData			:	ARRAY[0..4] OF WORD;
	StartHoldingWrite	:	BOOL;
	
	MBReadInputregs		:	FB_MBReadInputRegs;	//function 4
	InputRegData		:	ARRAY[0..27] OF WORD;
	StartInputRegRead	:	BOOL;
	
	MBReadInputs		:	FB_MBReadInputs;	//function 2
	InputData			:	ARRAY[0..2] OF BYTE;
	StartInputRead		:	BOOL;
	
	TransmissionDone	:	F_trig;
	bError				: BOOL;
	
	CommStep	:	UINT	:=	0;
	
	tpModbusDelay		: TP := (PT:= T#500MS);
END_VAR

tpModbusDelay();

IF NOT enable THEN
	commstep:= 0;
ELSIF (enable AND commstep = 0) THEN
	commstep := 1;
END_IF

MBWriteCoils(
	sIPAddr := set.IP,
	nTCPPort := 502,
	nUnitID := 1,//16#FF;
	nMBAddr := 0,//w_MBStartAddress,
	nQuantity := 50,
	cbLength := SIZEOF(CoilData),
	pSrcAddr := ADR(CoilData),
	bExecute := StartCoilWrite	//	<- werkt dit niet gewoon?
);

MBWriteHolding(
	sIPAddr := set.IP,
	nTCPPort := 502,
	nUnitID := 1,//16#FF;
	cbLength := SIZEOF(HoldingData),
	pSrcAddr := ADR(HoldingData),
	bExecute := StartHoldingWrite	//	<- werkt dit niet gewoon?
);
	
MBReadInputregs(
	sIPAddr := set.IP,
	nTCPPort := 502,
	nUnitID := 1,//16#FF;
	nMBAddr := 501,//w_MBStartAddress,
	nQuantity := 18,
	cbLength := SIZEOF(InputRegData),
	pDestaddr := ADR(InputRegData),
	bExecute := StartInputRegRead	//	<- werkt dit niet gewoon?
);

MBReadInputs(
	sIPAddr := set.IP,
	nTCPPort := 502,
	nUnitID := 1,//16#FF;
	nMBAddr := 501,//w_MBStartAddress,
	nQuantity := 5,
	cbLength := SIZEOF(InputData),
	pDestaddr := ADR(InputData),
	bExecute := StartInputRead	//	<- werkt dit niet gewoon?
);


CASE CommStep OF
	1: //Start MBWriteCoils
		CoilData[0].0 := set.GenOn = eOnoffState.Enable;
		CoilData[0].3 := set.GenOn = eOnoffState.Disable;
		
		CoilData[0].1 := set.GenBreakerOn = eOnoffState.Enable;
		CoilData[0].2 := set.GenBreakerOn = eOnoffState.Disable;
		
		CoilData[1].6 := set.GenAutoSyncOn = eOnoffState.Enable;
		CoilData[1].7 := set.GenAutoSyncOn = eOnoffState.Disable;
		
		CoilData[2].0 := set.bIslandModeEnable;
		CoilData[2].1 := set.bAMFModeEnable;
		CoilData[2].2 := set.bPeakshavingEnable;	
		CoilData[2].3 := set.bFixedPowerEnable;	
		CoilData[2].4 := set.bMPE;
		
		CoilData[3].0 := set.MainBreakerON = eOnoffState.Enable;
		CoilData[3].1 := set.MainBreakerON = eOnoffState.Disable;
		CoilData[3].2 := set.AutoStartStop;
		CoilData[3].3 := set.OperationMode = eGenOperationMode.ManualMode;
		CoilData[3].4 := set.OperationMode = eGenOperationMode.SemiAuto;	
		CoilData[3].5 := set.OperationMode = eGenOperationMode.Auto;	
		CoilData[3].6 := set.OperationMode = eGenOperationMode.Test;
		
		CoilData[6].0 := set.DroopEnable;
				
		StartCoilWrite := TRUE;
		Commstep := 2;
		
	2: //Wait for MBWriteCoils to finish
		StartCoilWrite := FALSE;
		bError := FALSE;
		IF NOT MBWriteCoils.bBusy THEN
			tpModbusDelay.IN := TRUE;
			IF NOT tpModbusDelay.Q THEN
				tpModbusDelay.IN := FALSE;
				IF NOT MBWriteCoils.bError THEN	
					Commstep := 3;
				 	//processdata
				ELSE
					//WriteFailed
					bError := TRUE;
					Commstep := 3;
				END_IF
			END_IF
		END_IF
		
	3: //Start MBWriteHolding
	 	MBWriteHolding.nMBAddr := 0;
		MBWriteHolding.nQuantity := 5;
		HoldingData[0] 	:= wordEndian(LIMIT(0, REAL_TO_UINT(set.Pset),100));
		HoldingData[1] 	:= wordEndian(LIMIT(60, REAL_TO_UINT(set.PFset),100));
		HoldingData[2] 	:= wordEndian(LIMIT(-100, REAL_TO_INT(set.Qset),100));
		HoldingData[3] 	:= wordEndian(LIMIT(-100, REAL_TO_INT(set.FreqRegulator),100));
		HoldingData[4] 	:= wordEndian(LIMIT(-100, REAL_TO_INT(set.VoltRegulator),100));
	
		StartHoldingWrite := TRUE;
		Commstep := 4;
		
	4: //Wait for MBWriteHolding to finish
		StartHoldingWrite := FALSE;
		
		IF NOT MBWriteHolding.bBusy THEN
			tpModbusDelay.IN := TRUE;
			IF NOT tpModbusDelay.Q THEN
				tpModbusDelay.IN := FALSE;
				IF NOT MBWriteHolding.bError THEN	
					Commstep := 5;
				 	//processdata
				ELSE
					//WriteFailed
					bError := TRUE;
					Commstep := 5;
				END_IF
			END_IF
		END_IF
		
	5: //Start MBReadInputregs
		StartInputRegRead := TRUE;
		Commstep := 6;
		
	6: //Wait for MBReadInputregs to finish
		StartInputRegRead := FALSE;
		IF NOT MBReadInputregs.bBusy THEN
			tpModbusDelay.IN := TRUE;
			IF NOT tpModbusDelay.Q THEN
				tpModbusDelay.IN := FALSE;
				IF NOT MBReadInputregs.bError THEN		
					get.ar_Linevoltage[phases.L1]	:= WORD_TO_REAL(WordEndian(InputRegData[0]));
					get.ar_Linevoltage[phases.L2]	:= WORD_TO_REAL(WordEndian(InputRegData[1]));
					get.ar_Linevoltage[phases.L3]	:= WORD_TO_REAL(WordEndian(InputRegData[2]));
					get.ar_LineVoltage[phases.AVG]	:= (get.ar_Linevoltage[phases.L1]+ get.ar_Linevoltage[phases.L2] + get.ar_Linevoltage[phases.L3]) / 3;
					
					get.ar_Phasevoltage[phases.L1]	:= WORD_TO_REAL(wordendian(InputRegData[3]));
					get.ar_Phasevoltage[phases.L2]	:= WORD_TO_REAL(wordendian(InputRegData[4]));
					get.ar_Phasevoltage[phases.L3]	:= WORD_TO_REAL(wordendian(InputRegData[5]));
					get.ar_PhaseVoltage[phases.AVG]	:= (get.ar_Phasevoltage[phases.L1]+ get.ar_Phasevoltage[phases.L2] + get.ar_Phasevoltage[phases.L3]) / 3;
							 
					get.ar_Frequency[phases.L1]		:= WORD_TO_REAL(wordendian(InputRegData[6])) / 100;
					get.ar_Frequency[phases.L2]		:= WORD_TO_REAL(wordendian(InputRegData[7])) / 100;
					get.ar_Frequency[phases.L3]		:= WORD_TO_REAL(wordendian(InputRegData[8])) / 100;
					get.ar_Frequency[phases.AVG]		:= (get.ar_Frequency[phases.L1]+ get.ar_Frequency[phases.L2] + get.ar_Frequency[phases.L3]) / 3;
							 
					get.ar_Current[phases.L1]	:= WORD_TO_REAL(wordendian(InputRegData[12]));
					get.ar_Current[phases.L2]	:= WORD_TO_REAL(wordendian(InputRegData[13]));
					get.ar_Current[phases.L3]	:= WORD_TO_REAL(wordendian(InputRegData[14]));
					get.ar_Current[phases.AVG] := (get.ar_Current[phases.L1] + get.ar_Current[phases.L2]  + get.ar_Current[phases.L3]) / 3;
						   
					get.ar_ActivePower[phases.L1]	:= WORD_TO_REAL(wordendian(InputRegData[15]));
					get.ar_ActivePower[phases.L2]	:= WORD_TO_REAL(wordendian(InputRegData[16]));
					get.ar_ActivePower[phases.L3]	:= WORD_TO_REAL(wordendian(InputRegData[17]));
					get.ar_ActivePower[phases.AVG]	:= (get.ar_ActivePower[phases.L1] + get.ar_ActivePower[phases.L2]  + get.ar_ActivePower[phases.L3]);
					
					Get.ar_ApparentPower[phases.AVG] := (get.ar_Current[phases.L1] * get.ar_PhaseVoltage[1] + get.ar_Current[phases.L2] * get.ar_PhaseVoltage[2] + get.ar_Current[phases.L3] * get.ar_PhaseVoltage[3]) / 1000;
					Get.ar_ReactivePower[phases.AVG] := ReactivePower(Get.ar_ApparentPower[phases.AVG], get.ar_ActivePower[phases.AVG], 0);  
					Get.ar_PowerFactor[phases.AVG] := PowerFactor(get.ar_ActivePower[phases.AVG],Get.ar_ApparentPower[phases.AVG], Get.ar_ReactivePower[phases.AVG]);
					Commstep := 7;
				ELSE
					//WriteFailed
					bError := TRUE;
					Commstep := 7;
				END_IF
			END_IF
		END_IF		
		
	7: //Start MBReadInputs
		StartInputRead := TRUE;
		Commstep := 8;
		
	8: //Wait for MBReadInputs to finish
		StartInputRead := FALSE;
		IF NOT MBReadInputs.bBusy THEN
			tpModbusDelay.IN := TRUE;
			IF NOT tpModbusDelay.Q THEN
				tpModbusDelay.IN := FALSE;
				IF NOT MBReadInputs.bError THEN
					get.bGenBreakerClosed 	:= InputData[0].0;  
					
					get.bMainBreakerClosed 	:= InputData[0].1;
					get.bGenRunning 		:= InputData[0].3;
					get.bGenVoltFreqOK 		:= InputData[0].4;
					get.bMainsFailure 		:= InputData[0].5;
					
					IF InputData[0].6 THEN	get.eActiveGenMode := eGenOperationMode.BlockMode;
					ELSIF InputData[0].7 THEN	get.eActiveGenMode := eGenOperationMode.ManualMode;
					ELSIF InputData[1].0 THEN	get.eActiveGenMode := eGenOperationMode.SemiAuto;
					ELSIF InputData[1].1 THEN	get.eActiveGenMode := eGenOperationMode.Auto;
					ELSIF InputData[1].2 THEN	get.eActiveGenMode := eGenOperationMode.Test;
					END_IF
					
					get.bIslandModeActive := InputData[1].5;
					get.bMainsFailure	:=	InputData[1].6;
					get.bPeakshaveActive := InputData[1].7;
					get.bFixedPowerActive := InputData[2].0;				
					Commstep := 9;
				ELSE
					//WriteFailed
					bError := TRUE;
					Commstep := 9;
				END_IF
			END_IF
		END_IF

	9: //Start MBWriteHolding
		MBWriteHolding.nMBAddr := 4125;
		MBWriteHolding.nQuantity := 1;
		HoldingData[0] 	:= wordEndian(LIMIT(0, REAL_TO_UINT(set.U_Fdroopset * 10), 100));

		StartHoldingWrite := TRUE;
		Commstep := 10;
		
	10: //Wait for MBWriteHolding to finish
		StartHoldingWrite := FALSE;
		
		IF NOT MBWriteHolding.bBusy THEN
			tpModbusDelay.IN := TRUE;
			IF NOT tpModbusDelay.Q THEN
				tpModbusDelay.IN := FALSE;
				IF NOT MBWriteHolding.bError THEN	
					Commstep := 1;
				 	//processdata
				ELSE
					//WriteFailed
					bError := TRUE;
					Commstep := 1;
				END_IF
			END_IF
		END_IF
END_CASE

ComOKRelease(IN:= NOT bError AND Commstep <>0, Q => get.CommunicationOK);

METHOD WordEndian : WORD
VAR_INPUT
	IN		: WORD;
END_VAR
IF b_changeEndianess THEN
	WordEndian := HOST_TO_BE16(IN);
ELSE
	WordEndian := IN;
END_IF
END_METHOD

END_FUNCTION_BLOCK

// ---- POUs/MAIN_Slow.TcPOU
PROGRAM MAIN_Slow
VAR
	{ attribute 'TcHmiSymbol.Hide' }
	monitor								: REFERENCE TO ST_System_Monitor;
	control								: ST_system_Control;
	
	{ attribute 'TcHmiSymbol.Hide' }				
	b_validref							: BOOL;
	Eventlog							: FB_Eventlogger;
	fbEventLogClient					: FB_EventLogClient;
	//InterMachineCom							: FB_InterMachineCommunication;
END_VAR

Errorhandling(b_ClearEvents := control.control.b_ClearHistory);

//Eventlogger instanciation
fbEventLogClient.Init(Eventlogger := Eventlog);
Eventlog(stparams:=Settings.MachineParams.Eventlogger, stParams := settings.MachineParams.Eventlogger);

//InterMachineCom(monitor:=monitor);
//Get refs of monitoring from fast cycle
monitor REF= MAIN_fast.monitor;
monitor.controlfb REF= control;


b_validref := __ISVALIDREF(monitor.powerstack) AND 
		__ISVALIDREF(monitor.battery) AND 
		__ISVALIDREF(monitor.neutraltransformer) AND
		__ISVALIDREF(monitor.powermonitor) AND
		__ISVALIDREF(monitor.protections) AND
		__ISVALIDREF(monitor.ACswitchgear) AND
		__ISVALIDREF(monitor.AcDcCharger) AND
		__ISVALIDREF(monitor.internalpsu) AND
		__ISVALIDREF(monitor.peakshavebox); // AND __ISVALIDREF(monitor)

IF b_validref THEN
	ControlManager(
		Monitor:=monitor,
		operation := control.Operation,
		control := control.control);
		control.HardSettings := ControlManager.PLCpersistvars.Hardsettings;
		control.SoftSettings := ControlManager.PLCpersistvars.Softsettings;

//VERY IMPORTANT. This closes the initialization after the slow cycle is executed the first time.
GVL.b_initCycle := FALSE;
END_IF

END_PROGRAM

// ---- POUs/Functions-FBs-Programs/FB_OverCurrentDetect.TcPOU
FUNCTION_BLOCK FB_OverCurrentDetect
VAR_INPUT
	ui_Ik					: UINT := 10; // kA/s 
	ui_RatedCurrent			: UINT; // A
	ui_gain					: UINT := 15;
	b_reset					: BOOL;
	r_In					: REAL;
	t_ResetTime				: TIME := T#2S;  
	t_MaxPickUpTime			: TIME := T#30M;
END_VAR
	
VAR_OUTPUT
	b_alarm						: BOOL;
	b_warning					: BOOL;
	ui_actLoad					: UINT; //%
	r_MaxCurrentDetected		: REAL;
	t_MaxTimeActive				: TIME;
	t_RemainingTime				: TIME;
END_VAR
VAR
	ton_PickUpTimer			: TON := (PT:=T#10S);
	ton_ResetTimer			: TON := (PT:=T#5S);
	r_MaxCurrent			: REAL;
	t_MaxTime				: TIME;
END_VAR

VAR
	r_ThermalMax		 	: REAL ;
	r_CurrentLimit			: REAL;
	r_Overcurrent			: REAL;
	r_thermalLoad			: REAL;
	r_thermalDelta			: REAL;
	r_thermalEnergy			: REAL;
	r_StepSize				: REAL;				
	//fb_loadMa				: FB_MovingAverage := (enable:= TRUE);
	i_instance				: INT;	
	init					: BOOL := TRUE;	
END_VAR

VAR_STAT
	i_instanceCounter		: INT;
	ton_evalTimer			: TON := (PT := T#10MS);
END_VAR

ton_pickUpTimer(PT:=t_MaxPickUpTime);
ton_ResetTimer(PT:=t_ResetTime);


IF i_instance = 0 THEN
	ton_EvalTimer(IN := NOT ton_evaltimer.Q);
END_IF

IF ton_evalTimer.Q THEN
	r_thermalMax := EXPT(TO_REAL(ui_Ik) * 1000,2);
	r_CurrentLimit := TO_REAL(ui_ratedCurrent);
	r_OverCurrent := r_in - r_CurrentLimit ;
	r_thermalLoad := EXPT(r_in, 2);
	r_StepSize := TO_REAL(ton_evalTimer.PT) / 1000;
	r_thermalDelta := EXPT(r_overcurrent * SEL(r_OverCurrent >0, ui_gain / 5, ui_gain),2) * SEL(r_OverCurrent >0, -1, 1);
	r_thermalEnergy := LIMIT(0, r_thermalEnergy + r_ThermalDelta * r_stepsize * 2, r_thermalMax * 1.01); // unknown why *2, but this gives correct remaining time...

	//fb_loadMa(IN := MAX(0,r_thermalDelta), Length := 2);
	
	IF r_IN >= r_CurrentLimit THEN
		t_remainingTime := MIN(t_maxPickUpTime - ton_pickUpTimer.ET, TO_TIME((MAX(0,r_thermalMax - r_thermalEnergy)) / MAX(1, r_thermalDelta) *1000)); 
		ui_actLoad := TO_UINT(r_In / MAX(1,ui_RatedCurrent) * 100);
		ton_PickUpTimer.IN := TRUE;
		ton_ResetTimer.IN := FALSE;
		IF t_MaxTime < ton_PickUpTimer.ET THEN
			t_MaxTime := ton_PickUpTimer.ET;
			t_MaxTimeActive := t_MaxTime;
		END_IF
		
		IF r_MaxCurrent < ABS(r_IN) THEN
			r_MaxCurrent := ABS(r_IN);
			r_MaxCurrentDetected := r_MaxCurrent;
		END_IF
	ELSIF r_IN < r_CurrentLimit THEN
		t_remainingTime := t_MaxPickUpTime;
		ton_ResetTimer.IN := TRUE;
		ton_PickUpTimer.IN := NOT(ton_ResetTimer.Q);
	END_IF
	
	b_Alarm := ton_PickUpTimer.Q OR t_remainingTime = T#0S;
	b_Warning := ton_PickUpTimer.IN;
	
	IF NOT ton_PickUpTimer.IN THEN
		ui_actLoad := 0;
		r_maxCurrent := 0;
		t_MaxTime := T#0S;
	END_IF
	
	IF b_reset THEN
		r_thermalEnergy := 0;
		r_MaxCurrentDetected := 0;
		t_MaxTimeActive := T#0S;
	END_IF

END_IF


IF init THEN
	init := FALSE;
	i_instance := i_instanceCounter;
	i_instanceCounter:= i_instanceCounter +1;
END_IF

END_FUNCTION_BLOCK

// ---- POUs/Functions-FBs-Programs/FB_UpperLimitAndTimeExceeded.TcPOU
FUNCTION_BLOCK FB_UpperLimitAndTimeExceeded
VAR_INPUT
	b_reset					: BOOL;
	r_In					: REAL;
	r_HighLimit				: REAL;
	r_Hysteresis			: REAL := 10;
	t_ResetTIME				: TIME;  
	t_PickUpTime			: TIME;
END_VAR
	
VAR_OUTPUT
	b_alarm						: BOOL;
	b_warning					: BOOL;
	r_MaxCurrentDetected		: REAL;
	t_MaxTimeActive				: TIME;
END_VAR
VAR
	ton_PickUpTimer			: TON := (PT:=T#10S);
	ton_ResetTimer			: TON := (PT:=T#5S);
	r_MaxCurrent			: REAL;
	t_MaxTime				: TIME;
END_VAR

ton_pickUpTimer(PT:=t_PickUpTime);
ton_ResetTimer(PT:=t_ResetTime);

IF r_IN >= r_HighLimit THEN
	ton_PickUpTimer.IN := TRUE;
	ton_ResetTimer.IN := FALSE;
	IF t_MaxTime < ton_PickUpTimer.ET THEN
		t_MaxTime := ton_PickUpTimer.ET;
		t_MaxTimeActive := t_MaxTime;
	END_IF
	
	IF r_MaxCurrent < ABS(r_IN) THEN
		r_MaxCurrent := ABS(r_IN);
		r_MaxCurrentDetected := r_MaxCurrent;
	END_IF
ELSIF r_IN < (r_HighLimit - r_Hysteresis) THEN
	ton_ResetTimer.IN := TRUE;
	ton_PickUpTimer.IN := NOT(ton_ResetTimer.Q);
END_IF

b_Alarm := ton_PickUpTimer.Q;
b_Warning := ton_PickUpTimer.IN;

IF NOT ton_PickUpTimer.IN THEN
	r_maxCurrent := 0;
	t_MaxTime := T#0S;
END_IF

IF b_reset THEN
	r_MaxCurrentDetected := 0;
	t_MaxTimeActive := T#0S;
END_IF

END_FUNCTION_BLOCK

// ---- POUs/Functions-FBs-Programs/_generalFunctions/PackByte.TcPOU
FUNCTION PackByte : INT
VAR_INPUT
	B0				: BOOL ;
	B1				: BOOL ;
	B2				: BOOL ;
	B3				: BOOL ;
	B4				: BOOL ;
	B5				: BOOL ;
	B6				: BOOL ;
	B7				: BOOL ;	
END_VAR
VAR
END_VAR

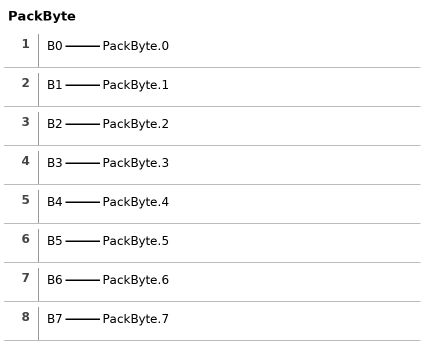
// NETWORK 1
PackByte.0 := B0;

// NETWORK 2
PackByte.1 := B1;

// NETWORK 3
PackByte.2 := B2;

// NETWORK 4
PackByte.3 := B3;

// NETWORK 5
PackByte.4 := B4;

// NETWORK 6
PackByte.5 := B5;

// NETWORK 7
PackByte.6 := B6;

// NETWORK 8
PackByte.7 := B7;

END_FUNCTION

// ---- POUs/Functions-FBs-Programs/_generalFunctions/XNOR.TcPOU
FUNCTION XNOR : BOOL
VAR_INPUT
	a : BOOL;
	b : BOOL;
END_VAR
VAR
END_VAR

XNOR := a AND b OR NOT (a OR b);

END_FUNCTION

// ---- POUs/Objects/DCLink/FB_ShuntBournsSSD.TcPOU
FUNCTION_BLOCK FB_ShuntBournsSSD
VAR	
	ReadInputs			: 	FB_MBReadRegs;
	InputData			:	ARRAY[0..20] OF WORD;
	StartReadinputs		:	BOOL;	
	InputReadError		:	Ton := (Pt := T#1S);
	dataInputs				: ARRAY[0..20] OF DWORD;
	lw_Power				: LWORD;  // Unsigned int32
	lw_Energy				: LWORD; // Unsigned int64
	lw_Coulomb				: LWORD; // Signed int64
	
	TON_UpdateInterval	:	Ton;
	
	State : UINT	:=	0;
	
END_VAR

VAR_INPUT
	b_enable				:	BOOL;
	IP				:	STRING	:= '192.168.1.65';
	UpdateInterval			:	TIME 	:=	T#100MS;
END_VAR

VAR_OUTPUT
	get					:	ST_Bourns_Powerdata;
	events				:	st_Bourns_errors;
	CommFault			:	Bool;
END_VAR

//Readinputs(
//	sIPAddr := IP,
//	nTCPPort := 502,
//	nUnitID := 1,
//	nMBAddr	:=	0,
//	nQuantity := 21,
//	cbLength := SIZEOF(InputData),
//	pDestAddr := ADR(InputData),
//	bExecute := StartReadinputs,
//);
//InputReadError();

//TON_UpdateInterval(in := NOT TON_UpdateInterval.Q);


//CASE State OF
//	0:
//		IF b_enable AND Ton_UpdateInterval.Q THEN
//			State := 10;
//		END_IF	
		
//	10:
//		StartReadInputs := TRUE;
//		state := 11;
		
//	11:
//		StartReadInputs := FALSE;
//		IF NOT ReadInputs.bBusy THEN
//			IF NOT ReadInputs.bError THEN
//				dataInputs[0]	:= SHL(WORD_TO_DWORD(InputData[1]), 16) OR (WORD_TO_DWORD(InputData[0]));   	
//				dataInputs[2]	:= SHL(WORD_TO_DWORD(InputData[3]), 16) OR (WORD_TO_DWORD(InputData[2])); 		
//				dataInputs[4]   := SHL(WORD_TO_DWORD(InputData[5]), 16) OR (WORD_TO_DWORD(InputData[4]));   
//				dataInputs[18]	:= SHL(WORD_TO_DWORD(InputData[19]), 16) OR (WORD_TO_DWORD(InputData[18]));	
				
//				lw_Coulomb 		:= SHL(WORD_TO_LWORD(InputData[9]), 48) OR SHL(WORD_TO_LWORD(InputData[8]), 32) OR 
//									SHL(WORD_TO_DWORD(InputData[7]), 16) OR (InputData[6]);								
//				lw_Power     		:= SHL(WORD_TO_DWORD(InputData[11]), 16) OR (WORD_TO_DWORD(InputData[10]));   	
//				lw_Energy 		:= SHL(WORD_TO_LWORD(InputData[15]), 48) OR SHL(WORD_TO_LWORD(InputData[14]), 32) OR 
//									SHL(WORD_TO_DWORD(InputData[13]), 16) OR (InputData[12]);							
	
//				get.Current			:= TO_REAL(DWORD_TO_DINT(dataInputs[0]))	/ 1000;  // mA to A
//				get.Temperature		:= TO_REAL(DWORD_TO_DINT(dataInputs[2])) / 10;	// 0.1 °C to °C
//				get.Voltage		   	:= TO_REAL(DWORD_TO_DINT(dataInputs[4])) / 1000; // mV to V
//				get.Power			:= TO_REAL(lw_Power) / 10000; // 0.1 W to kW	
//				get.Energy			:= TO_REAL(lw_Energy) / 1000;  // Wh to Kwh
				
//				events.b_OvervoltageError	:= DataInputs[16].0 OR DataInputs[16].6;
//				events.b_OverTemperatureError := DataInputs[16].4;
//				events.b_OverCurrentError := DataInputs[16].3 OR DataInputs[16].1;
//				events.b_EnergyOverflow		:= DataInputs[16].9;
//				events.b_DeviceFault		:= DataInputs[16].10 OR DataInputs[16].13 OR DataInputs[16].14 OR DataInputs[16].12;

//				InputReadError.IN := FALSE;
//			ELSE
//				InputReadError.IN := TRUE;
//			END_IF
//			State := 0;
//		END_IF

//END_CASE

//CommFault := inputReaderror.Q;

END_FUNCTION_BLOCK

// ---- POUs/Objects/PowerQualityMonitor/FB_EastronSDM630.TcPOU
FUNCTION_BLOCK FB_EastronSDM630 IMPLEMENTS ITF_StandardFB
VAR_INPUT
END_VAR
VAR_OUTPUT
END_VAR
VAR
	get			:	st_Eastron_get;	
END_VAR

Var_in_out constant
	st_params 	: 	st_EastronParams;
END_VAR

var	
	ReadInputRegs		:	FB_MBReadInputRegs;
	StartInputRegRead	:	Bool;
	InputRegData		:	Array[0..35] of dword;
	InputRegDataCommtimer	:	Ton := (PT := T#5s); 

	ReadInputRegsB			:	FB_MBReadInputRegs;
	StartInputRegReadB		:	Bool;
	InputRegDataB			:	Array[0..14] of dword;
	InputRegDataCommtimerB	:	Ton := (PT := T#5s); 	
	
	Step			: 	uint	:=	0;
		
	Ton_UpdateInterval	:	TON := (PT := T#1000ms);
	
	b_CommFault		:	Bool;
end_var



Ton_UpdateInterval(in := not Ton_UpdateInterval.Q);

InputRegDataCommtimer();
InputRegDataCommtimerB();

	
get.b_DataValid := not (InputRegDataCommtimer.Q or InputRegDataCommtimerB.q);
	
	case step of
		0:
			if Ton_UpdateInterval.Q then
				Step := 10;
			END_IF
				
		10: //read analog input status
			StartInputRegRead := true;	
			Step := 11;
		11: 
			StartInputRegRead := false;
			IF NOT ReadInputRegs.bBusy THEN
				IF NOT ReadInputregs.bError THEN	
					get.PhaseVoltage[phases.L1] := dWordToReal(InputRegData[0]);
					get.PhaseVoltage[phases.L2] := dWordToReal(InputRegData[1]);
					get.PhaseVoltage[phases.L3] := dWordToReal(InputRegData[2]);
					
					get.Current[phases.L1] := dWordToReal(InputRegData[3]);
					get.Current[phases.L2] := dWordToReal(InputRegData[4]);
					get.Current[phases.L3] := dWordToReal(InputRegData[5]);
					
					get.ActivePower[phases.L1] := dWordToReal(InputRegData[6]);
					get.ActivePower[phases.L2] := dWordToReal(InputRegData[7]);
					get.ActivePower[phases.L3] := dWordToReal(InputRegData[8]);
					
					get.ApparentPower[phases.L1] := dWordToReal(InputRegData[9]);
					get.ApparentPower[phases.L2] := dWordToReal(InputRegData[10]);
					get.ApparentPower[phases.L3] := dWordToReal(InputRegData[11]);
					
					get.ReactivePower[phases.L1] := dWordToReal(InputRegData[12]);
					get.ReactivePower[phases.L2] := dWordToReal(InputRegData[13]);
					get.ReactivePower[phases.L3] := dWordToReal(InputRegData[14]);
					
					get.Powerfactor[phases.L1] := dWordToReal(InputRegData[15]);
					get.Powerfactor[phases.L2] := dWordToReal(InputRegData[16]);
					get.Powerfactor[phases.L3] := dWordToReal(InputRegData[17]);
					
					get.PhaseVoltage[phases.AVG] 	:= dWordToReal(InputRegData[21]);
					get.Current[phases.avg] 		:= dWordToReal(InputRegData[23]);
					get.ActivePower[phases.Sum] 	:= dWordToReal(InputRegData[26]);
					get.ApparentPower[phases.Sum] 	:= dWordToReal(InputRegData[28]);	
					get.ReactivePower[phases.Sum] 	:= dWordToReal(InputRegData[30]);
					get.Powerfactor[phases.AVG] 	:= dWordToReal(InputRegData[31]);	
					
					get.Frequency					:= dWordToReal(InputRegData[35]);
					
					InputRegDataCommtimer.in := false;
				else
					InputRegDataCommtimer.IN := true;
				END_IF
				step := 20;
			end_if
			
		20: //read analog input status
			StartInputRegReadB := true;	
			Step := 21;
		21: 
			StartInputRegReadB := false;
			IF NOT ReadInputRegsB.bBusy THEN
				IF NOT ReadInputregsB.bError THEN	
					get.TotalActiveEnergyIn[phases.L1] := dWordToReal(InputRegDataB[0]);
					get.TotalActiveEnergyIn[phases.L2] := dWordToReal(InputRegDataB[1]);
					get.TotalActiveEnergyIn[phases.L3] := dWordToReal(InputRegDataB[2]);
					get.TotalActiveEnergyIn[phases.Sum] := get.TotalActiveEnergyIn[phases.L1] + get.TotalActiveEnergyIn[phases.L2] + get.TotalActiveEnergyIn[phases.L3];
					
					get.TotalActiveEnergyOut[phases.L1] := dWordToReal(InputRegDataB[3]);
					get.TotalActiveEnergyOut[phases.L2] := dWordToReal(InputRegDataB[4]);
					get.TotalActiveEnergyOut[phases.L3] := dWordToReal(InputRegDataB[5]);
					get.TotalActiveEnergyOut[phases.Sum] := get.TotalActiveEnergyOut[phases.L1] + get.TotalActiveEnergyOut[phases.L2] + get.TotalActiveEnergyOut[phases.L3];

					get.TotalReactiveEnergyIn[phases.L1] := dWordToReal(InputRegDataB[9]);
					get.TotalReactiveEnergyIn[phases.L2] := dWordToReal(InputRegDataB[10]);
					get.TotalReactiveEnergyIn[phases.L3] := dWordToReal(InputRegDataB[11]);
					get.TotalReactiveEnergyIn[phases.Sum] := get.TotalReactiveEnergyIn[phases.L1] + get.TotalReactiveEnergyIn[phases.L2] + get.TotalReactiveEnergyIn[phases.L3];
					
					get.TotalReActiveEnergyOut[phases.L1] := dWordToReal(InputRegDataB[12]);
					get.TotalReActiveEnergyOut[phases.L2] := dWordToReal(InputRegDataB[13]);
					get.TotalReActiveEnergyOut[phases.L3] := dWordToReal(InputRegDataB[14]);
					get.TotalReActiveEnergyOut[phases.Sum] := get.TotalReActiveEnergyOut[phases.L1] + get.TotalReActiveEnergyOut[phases.L2] + get.TotalReActiveEnergyOut[phases.L3];
					
					InputRegDataCommtimerB.in := false;
				else
					InputRegDataCommtimerB.in := True;
				END_IF
				step := 0;
			end_if			
	END_CASE


ReadInputregs(
	sIPAddr := st_params.IPaddress,
	nTCPPort := 502,
	nUnitID := 1,
	nMBAddr := 0,
	nQuantity := 72,
	cbLength := SIZEOF(InputRegData),
	pDestaddr := ADR(InputRegData),
	bExecute := StartInputRegRead	
);

ReadInputregsB(
	sIPAddr := st_params.IPaddress,
	nTCPPort := 502,
	nUnitID := 1,
	nMBAddr := 173,
	nQuantity := 28,
	cbLength := SIZEOF(InputRegDataB),
	pDestaddr := ADR(InputRegDataB),
	bExecute := StartInputRegReadB	
);

METHOD DwordToReal : Real
VAR_INPUT
	in	:	Dword;
END_VAR

var
	DwToReal	:	un_WordToFloat;
	RealVar		:	real;
END_VAR
dWToReal.dwordVal := BE32_to_host(in);
RealVar := DwToReal.floatVal;

if not isNAN(RealVar) then
	DwordToReal := RealVar;
END_IF
END_METHOD

{warning 'Add method implementation '}
METHOD EMstop : BOOL
END_METHOD

{warning 'Add method implementation '}
METHOD getDiagnostics
VAR_INPUT
	AddError	: POINTER TO FB_AddErrorST;
	a_ActiveEvents	: POINTER TO ST_ErrorStruct;
END_VAR
VAR_IN_OUT
	w_Index	: WORD;
END_VAR
END_METHOD

{warning 'Add method implementation '}
METHOD Init : BOOL
END_METHOD

{warning 'Add method implementation '}
METHOD Reset : BOOL
END_METHOD

END_FUNCTION_BLOCK

// ---- POUs/Objects/InterMachineCom/FB_ConnectMqttBroker.TcPOU
FUNCTION_BLOCK FB_ConnectMqttBroker
VAR_INPUT
	bRestartConnection			: BOOL;
	bConnect					: BOOL;
	sHostName					: STRING;
					
END_VAR
VAR_OUTPUT
	eConnectionState			: eConnectionState;
	bIncomingMsg	: BOOL;
	sMessage		: STRING;
END_VAR
VAR
	fbMqttClient					: FB_IotMqttClient;
	fbMessageQueue					: FB_IotMqttMessageQueue;
	fbMessage						: FB_IotMqttMessage;
	ton_ReconnectionTimer			: TON := (PT:=T#5S);
	bSetParameter					: BOOL;
	rTrigReinitCom					: R_TRIG;
	rTrigComStateOK					: R_Trig;
	
	//subscription
	bSubscribed 					: BOOL;
	sSubscribedTopic 				: STRING;
	sReceivedTopic					: STRING;
	
	//json files
	fbJson         	: FB_JsonSaxWriter;
  	fbJsonDataType 	: FB_JsonReadWriteDataType;
	sJsonDocPub     : STRING(255);
END_VAR

ton_ReconnectionTimer(IN:= NOT ton_ReConnectionTimer.Q AND NOT fbMqttClient.bConnected);
rTrigReinitCom(CLK := bRestartConnection);
bIncomingMsg := FALSE;

IF ton_reconnectionTimer.Q OR rTrigReinitCom.Q THEN
	eConnectionState := eConnectionState.disconnected;
	//Reset connection
	fbMqttClient.Execute(FALSE);
	//Configure
	IF bSetParameter THEN
		bSetParameter := FALSE;
		fbMqttClient.sHostName							:= sHostName;
		fbMqttClient.nHostPort							:= 1883;
		fbMqttClient.ipMessageQueue						:= fbMessageQueue;
	END_IF
ELSE
	fbMqttClient.Execute(bConnect);
	//Reset parameter set for next time connecting
	bSetParameter := TRUE;
END_IF

rTrigComStateOK(CLK := fbMqttClient.bConnected);
IF rTrigComStateOK.Q THEN
	eConnectionState := eConnectionState.connected;
END_IF


//receive message at subscribed topic
IF fbMessageQueue.nQueuedMessages > 0 THEN
	 IF fbMessageQueue.Dequeue(fbMessage:=fbMessage) THEN
		fbMessage.GetTopic(pTopic:=ADR(sReceivedTopic), nTopicSize:=SIZEOF(sReceivedTopic) );
			// Process asset messages
			bIncomingMsg	:= TRUE;
			fbMessage.GetPayload(pPayload:=ADR(sMessage), nPayloadSize:=SIZEOF(sMessage), bSetNullTermination:=TRUE);
			sMessage:=LEFT(sMessage,LEN(sMessage) -1 );
	END_IF
END_IF

//TO ADD, when no slaves are present, reduce publish interval

METHOD Publish : BOOL
VAR_INPUT
	Interval		: TIME;
	sTopic			: STRING;
	sMessage		: STRING;
END_VAR

VAR_INST
	tMinInterval 				: TIME := T#10MS;
	tonPublishInterval			: TON;
END_VAR
// publish
tonpublishInterval(PT := MAX(tMinInterval, Interval));

IF fbMqttClient.bConnected THEN
    tonPublishInterval.IN := TRUE;
    IF tonPublishInterval.Q THEN // publish new payload every second
        tonPublishInterval.IN := FALSE;
		fbMqttClient.Publish(sTopic:=sTopic,
		pPayload := ADR(sMessage),
		nPayloadSize := LEN2(ADR(sMessage)),
		eQoS := TcIotMqttQos.AtMostOnceDelivery,
		bRetain:= FALSE,
		bQueue := FALSE);
    END_IF
END_IF
END_METHOD

METHOD Subscribe : BOOL;
VAR_INPUT
	sTopic		: STRING; 
END_VAR

VAR_INST
	sReceivedTopic : STRING;
END_VAR
IF fbMqttClient.bConnected AND NOT bSubscribed THEN
	sSubscribedTopic := sTopic;
   bSubscribed := fbMqttClient.Subscribe(sTopic:=sTopic, eQoS:=TcIotMqttQos.AtMostOnceDelivery); //sSubTopic
END_IF

IF sSubscribedTopic <> sTopic THEN
	bSubscribed := FALSE;
END_IF
END_METHOD

END_FUNCTION_BLOCK

// ---- POUs/Objects/InterMachineCom/FB_InterMachineCommunication.TcPOU
FUNCTION_BLOCK FB_InterMachineCommunication
VAR_INPUT
	SlaveConnectionData				: ST_InterMachineCom_SlaveConData;

END_VAR

VAR_IN_OUT CONSTANT
	monitor							: ST_system_monitor;
	st_params						: ST_InterMachineCom_Params;
END_VAR

VAR_IN_OUT
	control							: ST_system_control;
END_VAR

VAR_OUTPUT
	e_state							: eConnectionState;
END_VAR

VAR
	InternalBroker					: FB_ConnectMqttBroker;
	ExternalBroker					: FB_ConnectMQttBroker;
	
	bSetParameter					: BOOL;
	bConnect						: BOOL := TRUE;
	bIncommingMsg					: BOOL;
	hrErrorOccurred 				: DINT; //Contains latest error message
	sTopicRec						: STRING(255);
	sMessage						: STRING(255);
	ReinitComParams					: BOOL;
	
	
	bSubscribed						: BOOL;
	ton_PublishInterval				: TON;
	sPubTopic						: STRING;
	sSubTopic						: STRING;
	
	stPubDataMaster					: ST_InterMachineCom_Master;
	stPubDataSlave					: st_InterMachineCom_Slave;
	stSubDataMaster					: ST_InterMachineCom_Master;
	stSubDataSlave					: st_InterMachineCom_Slave;
	
	
	fbJson         	: FB_JsonSaxWriter;
  	fbJsonDataType 	: FB_JsonReadWriteDataType;
	sJsonDocPub     : STRING(255);
	bRecJsonOK		: BOOL;
	
	
	sMasterTopic 	: STRING := 'master';
END_VAR

(* 
Internal broker is used to post local data in the master topic. The unit listens to the slave topics

*)

//Connect brokers

//Generate machinedata for internal master
InternalBroker(bConnect := TRUE, sHostname := ST_params.InternalBrokerIP);
InternalBroker.Publish(
	Interval := st_params.MasterPublishRate, 
	sTopic := sMasterTopic, 
	sMessage := StructToJson(TRUE));
InternalBroker.Subscribe(sTopic := 'slave/epu/#/read');

IF internalbroker.bIncomingMsg THEN
	JsonToStruct(sMessage := internalbroker.sMessage);
END_IF

//Generate slave data for the external master
ExternalBroker(bConnect := SlaveConnectionData.enable, sHostname := SlaveConnectionData.BrokerIP);
ExternalBroker.Publish(Interval := st_params.SlavePublishRate, 
		sTopic := CONCAT(CONCAT('epu/slave/',settings.Properties.s_SerialNumber),'/read'),
		sMessage := StructToJson(FALSE));
ExternalBroker.Subscribe(sTopic := sMasterTopic);

IF Externalbroker.bIncomingMsg THEN
	JsonToStruct();
END_IF




//Publish as master 
sPubTopic := 'master';
sSubTopic := 'slave/#';
//Ton_PublishInterval.PT := st_params.MasterPublishRate;
//generate json doc
fbJson.ResetDocument();
fbJsonDataType.AddJsonValueFromSymbol(fbJson, 'ST_InterMachineCom_Master', SIZEOF(stPubDataMaster), ADR(stPubDataMaster));
fbJson.EndObject();
fbJson.CopyDocument(sJsonDocPub, SIZEOF(sJsonDocPub));

IF SlaveConnectionData.enable AND SlaveConnectionData.BrokerIP <> '' THEN
	sSubTopic := 'master';
	sPubTopic := CONCAT('slave/', settings.Properties.s_SerialNumber);
	Ton_PublishInterval.PT := st_params.MasterPublishRate;
	//generate json doc
	fbJson.ResetDocument();
	fbJsonDataType.AddJsonValueFromSymbol(fbJson, 'ST_InterMachineCom_Slave', SIZEOF(stPubDataSlave), ADR(stPubDataSlave));
	fbJson.EndObject();
	fbJson.CopyDocument(sJsonDocPub, SIZEOF(sJsonDocPub));
	
	//converter receiving message back to structur
	fbJsonDataType.SetSymbolFromJson(sMessage, 'st_InterMachineCom_Master', SIZEOF(stSubDataMaster), ADR(stSubDataMaster));
END_IF

// publish
IF fbMqttClientInternal.bConnected THEN
    IF NOT bSubscribed THEN
        bSubscribed := fbMqttClientInternal.Subscribe(sTopic:=sSubTopic, eQoS:=TcIotMqttQos.AtMostOnceDelivery); //sSubTopic
    END_IF
    ton_PublishInterval(IN:=TRUE);
    IF ton_PublishInterval.Q THEN // publish new payload every second
        ton_PublishInterval(IN:=FALSE);
			fbMqttClientInternal.Publish(sTopic:=sPubTopic,
			pPayload := ADR(sJsonDocPub),
			nPayloadSize := LEN2(ADR(sJsonDocPub)),
			eQoS := TcIotMqttQos.AtMostOnceDelivery,
			bRetain:= TRUE,
			bQueue := FALSE);
    END_IF
END_IF


IF bIncommingMsg THEN
	bRecJsonOK := fbJsonDataType.SetSymbolFromJson(sMessage, 'st_InterMachineCom_Slave', SIZEOF(stSubDataSlave), ADR(stSubDataSlave));
END_IF

Internalbroker.Subscribe();

METHOD CheckSlaves : BOOL
VAR_INPUT
END_VAR
END_METHOD

METHOD GetSubData : BOOL
VAR_INPUT
END_VAR
END_METHOD

METHOD JsonToStruct : BOOL
VAR_INPUT
	MasterMode		: BOOL;
END_VAR

VAR_IN_OUT
	sMessage : STRING;
END_VAR
IF MasterMode THEN
	//Get the message from the external broker 'master' subscribtion, format according to ST_IntermachineCom_Master
ELSE
	//Get the message from the internal broker '+/slave/#/read' subscriptiom, format according to ST_intermachineCom_Slave
	(* A json parser need to be constructed such that the combined json struct is formatted in separate st_IntermachineCom_slave structs.
	
	Data can come from the epu or hpu and distinquish is made through the topic path: /slave/hpu/#, or /slave/epu/#
	For example the epu slave path is: /slave/epu/{serialnumber}/read and the ST_intermachineCom_slave struct comes out.
	A json filter has to be made to iterate along all serial numbers in epu and hpu group. 
	A method must be created where the data is temporarily stored such that the ACP (available charge power), 
	ADP (available discharge power) and ARP (available reactive power) can me summed and used for the power setpoint calculation.
	
	A separate topic /slave/epu/{serialnumber}/write can be used to control slaves individually with the ST_IntermachineCom_master struct.
	However, this requires the slave CW heartbeat and SW heartbeat to be updated within heartbeat time limit. When the CW heartbeat stops, 
	the slave will go to general operation related to the 'master' topic that is broadcasted. 
	*)
END_IF
END_METHOD

METHOD Reset : BOOL
VAR_INPUT
END_VAR
IF InternalBroker.bRestartConnection AND ExternalBroker.bRestartConnection THEN
	InternalBroker.bRestartConnection := FALSE;
	ExternalBroker.bRestartConnection := FALSE;
	Reset := TRUE;
ELSE
	InternalBroker.bRestartConnection := NOT InternalBroker.bRestartConnection;
	ExternalBroker.bRestartConnection := NOT ExternalBroker.bRestartConnection;
END_IF
END_METHOD

METHOD SetPubData : BOOL
VAR_INPUT
END_VAR

VAR_INST
	WatchdogPulse	: TON; 
END_VAR
WatchdogPulse(IN := NOT watchdogPulse.Q, PT:= st_params.WatchdogPulseRate);

//Internal 'master' data to control slaves
stPubDataMaster.CW.0 := monitor.powerstack.b_StartedState;
stPubDataMaster.CW.1 := monitor.powerstack.e_State = eStatusPowerstack.idle;
stPubDataMaster.CW.2 := monitor.powerstack.e_State = eStatusPowerstack.shutdown;
stPubDataMaster.CW.3 := GVL.b_EmergencyShutdownActive AND ST_IntermachineCom_params.EMstopCoupling;
stPubDataMaster.CW.4 := monitor.system.e_State = eSystemState.Reset;
stPubDataMaster.CW.15 := SEL(watchdogPulse.Q, stPubDataMaster.CW.15, NOT stPubDataMaster.CW.15);
stPubDataMaster.PS := 0; // TBD based on slaves
stPubDataMaster.QS := 0; 

//Slave data for external master
stPubDataSlave.ACP := TO_UINT(ABS(monitor.powerstack.r_Pmin));
stPubDataSlave.ADP := TO_UINT(ABS(monitor.powerstack.r_PMax));
stPubDataSlave.AQ := TO_UINT(ABS(monitor.powerstack.r_QMax));
stPubDataSlave.SW.0 := monitor.system.e_State = eSystemState.StandBy OR monitor.system.e_State = eSystemState.Conditioning;
stPubDataSlave.SW.1 := monitor.powerstack.b_StartedState;
stPubDataSlave.SW.2 := monitor.system.e_State = eSystemState.Stopped;
stPubDataSlave.SW.3 := monitor.system.e_State = eSystemState.Discharging_Only;
stPubDataSlave.SW.4 := monitor.system.e_State = eSystemState.Charging_Only;
stPubDataSlave.SW.5 := GVL.b_WarningActive;
stPubDataSlave.SW.6 := GVL.b_NormalShutdownActive;
stPubDataSlave.SW.7 := GVL.b_EmergencyShutdownActive;
stPubDataSlave.SW.15 := stSubDataMaster.CW.15;
END_METHOD

METHOD StructToJson : STRING
VAR_INPUT
	Mastermode		: BOOL; //if false, then slave mode
END_VAR
fbJson.ResetDocument();

IF MasterMode THEN
	fbJsonDataType.AddJsonValueFromSymbol(fbJson, 'ST_InterMachineCom_Master', SIZEOF(stPubDataMaster), ADR(stPubDataMaster));
ELSE
	fbJsonDataType.AddJsonValueFromSymbol(fbJson, 'ST_InterMachineCom_Slave', SIZEOF(stPubDataSlave), ADR(stPubDataSlave));
END_IF

fbJson.EndObject();
fbJson.CopyDocument(StructToJson, SIZEOF(StructToJson));
END_METHOD

END_FUNCTION_BLOCK

// ---- POUs/Objects/PLCStatus/FB_PLCUpdate.TcPOU
FUNCTION_BLOCK FB_PLCUpdate

VAR_INPUT
	bUpdate				: BOOL;
	bAbortUpdate		: BOOL;
END_VAR

VAR_OUTPUT
	FTPState			: eFTPstate;
	InstalState			: eInstalState;
	BackupState			: eInstalState;
	sLogMessage 		: STRING(255);
	bCheckUpdates		: BOOL;	
	bUpdateAvailable 	: BOOL;
END_VAR

VAR	
	rTrig_CheckUpdate	: R_Trig;
	
    fbFileDelete 		: FB_FileDelete;  (* Om oude bestanden te verwijderen *)
    
    sJsonUrl      		: STRING := 'http://server.com/updates.json'; (* JSON met update-info *)
    sUpdateUrl    		: STRING := '';  (* URL van het updatebestand uit JSON *)
    sLocalPath    		: STRING := '/usr/local/updates/update.tsmpkg';
    sBackupPath   		: STRING := '/usr/local/backup/old_version.tsmpkg';
    
    sCurrentVersion 	: STRING := '1.2.0';  (* Huidige versie van de PLC *)
    sNewVersion     	: STRING := '';       (* Nieuwe versie uit JSON *)

   
    bDownloadComplete 	: BOOL;
    bInstallComplete 	: BOOL;
    bRollbackNeeded 	: BOOL;
    eState 				: INT := 0;
    iRetryCount 		: INT := 0;
END_VAR




CASE eState OF
    0: // Controleer op update via JSON
		rTrig_CheckUpdate(CLK := bUpdate);
		IF rTrig_CheckUpdate THEN
			bCheckUpdates := TRUE;
		END_IF
		
		IF 
		CheckForUpdates();
        

    1: // Maak een backup van de huidige versie
		BackupState := Copy(sSrcPath := sLocalPath, sDestPath := sBackupPath);
		
        IF BackupState = eInstalState.Success THEN
            eState := 2;
		ELSIF BackupState = eInstalState.Failure OR bAbortUpdate THEN
			eState := 99;
        END_IF

    2: // Download de nieuwe update via FTP
		FTPState := DownloadUpdate(
			sHost := 'temp',
			sUsername := 'tempuser',
			sPassword := 'tempPass',
			sSrcFile := 'path/1',
			sDesFile := 'path/2',
			start :=  bUpdateAvailable);

        IF FTPState = eFTPState.Success THEN
            bDownloadComplete := TRUE;
            eState := 3;
        ELSIF FTPState = eFTPState.Failure OR bAbortUpdate THEN
                eState := 99; // Ga naar fallback
        END_IF

    3: // Wachten op bevestiging van de gebruiker via HMI
        IF bUpdate THEN
			bUpdateStarted := TRUE;
            eState := 4;
        END_IF

    4: // Installeer de update
		InstalState := Copy(sSrcPath := sLocalPath, sDestPath := 'path/2');
		IF InstalState = eInstalState.Success THEN
			bInstallComplete := TRUE;
			eState := 5;
		ELSIF InstalState = eInstalState.Failure OR bAbortUpdate THEN
			bRollbackNeeded := TRUE;
            eState := 6; // Ga naar rollback
		END_IF

    5: // Herstart de PLC na succesvolle update
        SystemReboot();

    6: // Rollback uitvoeren als de update is mislukt
		InstalState := Copy(sSrcPath := sBackupPath,  sDestPath := '/usr/local/boot/update.tsmpkg');

		IF InstalState = eInstalState.Success THEN
			SystemReboot();  // Herstart de PLC met oude versie
		ELSIF InstalState = eInstalState.Failure OR bAbortUpdate THEN
			eState := 99;  // Fallback activeren als rollback mislukt
		END_IF

    99: // Fallback: Stop het updateproces en meld de fout
        bUpdateAvailable := FALSE;
		bUpdateStarted := FALSE;
        bRollbackNeeded := FALSE;
        iRetryCount := 0;
END_CASE

CASE eState OF
    0:	sLogMessage := 'Check if update is available';
        WriteLog(sLogMessage);
        
   1:	sLogMessage := 'Create backup of current software';
        WriteLog(sLogMessage);

    2:	sLogMessage := 'Downloading update';
        WriteLog(sLogMessage);
		
	3:	sLogMessage := 'Update ready for installation';
		WriteLog(sLogMessage);
		
	4:	sLogMessage := 'Installing update';
		WriteLog(sLogMessage);
		
	5:	sLogMessage := 'Rebooting system';
		WriteLog(sLogMessage);    
		
    6:	sLogMessage := 'Update failed, rollback started';
         WriteLog(sLogMessage);
		 
    99:
        sLogMessage := 'Update mislukt, fallback geactiveerd';
        WriteLog(sLogMessage);
END_CASE

METHOD CheckForUpdates : BOOL
VAR_INPUT
	sServerUrl   : STRING := 'http://server.com/updates.json'; (* Volledige URL *)
END_VAR

VAR_INST
	fbHttpClient 		: FB_IotHttpClient;  (* Voor JSON versiecontrole *)
	     
    sResponse    : STRING(1024);  (* Buffer voor de server response *)
    bExecute     : BOOL := TRUE;
    bDone        : BOOL;
    bError       : BOOL;
END_VAR
fbHttpClient(
	sHostName := sHostName,
	


fbHttpClient.sHost := 'server.com';  // Vervang met je eigen server
fbHttpClient.sResource := '/updates.json';  // JSON-bestand
fbHttpClient.eMethod := E_HttpMethod.GET;
fbHttpClient.bExecute := TRUE;

IF fbHttpClient.eState = E_HttpRequestState.Done THEN
	sNewVersion := ExtractJsonValue(fbHttpClient.sResponseContent, 'latest_version');
	sUpdateUrl := ExtractJsonValue(fbHttpClient.sResponseContent, 'update_file');
	
	IF sNewVersion > sCurrentVersion THEN
		bUpdateAvailable := TRUE;
		eState := 1;
	END_IF
END_IF


(* Stap 1: HTTP Request starten *)
IF bExecute THEN
    fbHttpClient. := sServerUrl;   (* Geef de volledige URL mee *)
    fbHttpClient.eMethod := T_IotHttpMethod.Get;  (* HTTP GET Methode *)
    fbHttpClient.bExecute := TRUE;
    bExecute := FALSE; (* Voorkomt dat het telkens opnieuw start *)
END_IF

(* Stap 2: Wachten op antwoord *)
IF fbHttpClient.bDone THEN
    sResponse := fbHttpClient.sResponse;  (* Server response opslaan *)
    bDone := TRUE;
ELSIF fbHttpClient.bError THEN
    bError := TRUE;
END_IF
END_METHOD

METHOD Copy : eInstalstate
VAR_INPUT
	sSrcPath : STRING;
	sDestPath: STRING;
END_VAR

VAR_OUTPUT
	Busy 		: BOOL;
    Error 		: BOOL;
	ErrID 		: UDINT;
END_VAR

VAR_INST
	ton_waitRetry		: ton := (pt := T#2S);
	fbFileCopy   		: FB_FileCopy;    (* Voor het maken van een backup *)
END_VAR
fbFileCopy(
	sSrcPathName := sSrcPath,
	sDestPathName := sDestPath,
	tTimeOut := T#15S,
	bBusy => Busy,
	bError => Error,
	nErrId => ErrID);
	
ton_waitRetry(Q => fbFileCopy.bExecute);

IF Error THEN
	Copy := eInstalState.Failure;
ELSIF busy THEN
	Copy := eInstalState.InProgress;
	ton_waitRetry.IN := FALSE;
ELSE
	IF NOT fbFileCopy.bExecute THEN
		Copy := eInstalState.Success;
	END_IF
	ton_waitRetry.IN := TRUE;
END_IF
END_METHOD

METHOD DownloadUpdate : eFTPState

VAR_INPUT
	sHost 			: STRING := 'ftp.example.com';
	sUsername		: STRING;
	sSrcFile		: STRING;
	sDesFile		: STRING;
	sPassword		: STRING;
	Start			: BOOL;
END_VAR

VAR_OUTPUT
	Busy 		: BOOL;
    Error 		: BOOL;
	ErrID 		: UDINT;
END_VAR

VAR_INST
	bRetry			: BOOL;
	byMaxRetries	: BYTE := 3;
	byRetryCounter	: BYTE;
	StartTrigger : R_TRIG;	
	FTPstate 	: eFTPState;
	ftpOpen 	: FB_FTP_Open; 			// Function block om verbinding te openen.
	ftpDownload : FB_FTP_FileDownload; 	// Function block om het bestand te downloaden
    ftpClose 	: FB_FTP_Close;  			// Function block om de verbinding te sluiten
    hFTP 		: T_HFTP; //FTP handle / identifyer
	RTrig_Error	: R_Trig;
END_VAR
StartTrigger(CLK:= start);

CASE FTPState OF
      eFTPState.Disconnected:
			IF StartTrigger.Q OR bRetry THEN
				bRetry := FALSE;
      			FTPState := eFTPState.Connecting;
			END_IF
			
     eFTPState.Connecting:
         ftpOpen(
			sHost:= sHost,
			nPort:= 21,
			sUsername:= sUsername,
			sPassword:= sPassword,
			tTimeout:= T#15S,
			bExecute := TRUE,
			hFTP=> hFTP,
			bBusy => busy,
			bError => Error,
			nErrID=> ErrID
			);
         IF NOT Busy AND NOT Error THEN
             ftpOpen(bExecute:= FALSE);
             FTPState := eFTPstate.Downloading;
         END_IF
		 
     eFTPstate.Downloading:
		ftpDownload(
			sNetID:= '',              // Lokale machine
			hFTP:= hFTP,              // Gebruik de handle van de geopende verbinding
			sSrcFile:= '\TestFolder\File1.txt',
            sDesFile:= '\Program Files\TestFile1.txt',
			tTimeout:= T#15S,         // Timeout
			bexecute := TRUE,
			bBusy => busy,
            bError => error,
			nErrID=> ErrID
		);
         IF NOT busy AND NOT Error THEN
             ftpDownload(bExecute:= FALSE);
             FTPState := eFTPState.Success;
         END_IF
     eFTPState.Success:
		ftpClose(
			sNetID:= '',              // Lokale machine
			hFTP:= hFTP,              // Gebruik de handle van de geopende verbinding
			bExecute:= TRUE,      // Start het sluiten van de verbinding
			bBusy => busy,
            bError => error,
			tTimeout:= T#15S,         // Timeout
			nErrID=> ErrID
		);
	 	
       	 IF NOT busy AND NOT Error THEN
             ftpClose(bExecute:= FALSE);
             FTPstate := eFTPState.Disconnected;
			 byRetryCounter := 0;
         END_IF
		
	eFTPState.Failure:
		IF StartTrigger.Q THEN
			FTPState := eFTPState.Connecting;
		END_IF	 	
END_CASE

//Retry on error trigger
RTrig_Error(CLK:= Error);
IF RTrig_Error.Q THEN
	IF ByRetryCounter < byMaxRetries THEN
		FTPstate := eFTPState.Disconnected;
		bRetry := TRUE;
		byRetryCounter := byRetryCounter +1;
	ELSE
		FTPstate := eFTPState.Failure;
	END_IF
END_IF

DownloadUpdate := FTPState;
END_METHOD

METHOD SystemReboot : BOOL
VAR_INPUT
END_VAR

VAR_INST
    fbSysRestart 		: TC_Restart; (* Systeemherstartfunctie *)
END_VAR
fbSysRestart();
END_METHOD

METHOD WriteLog : BOOL
VAR_INPUT
    sMessage : STRING;
END_VAR

VAR_INST
    fbLogWriter 		: FB_FileWrite;
END_VAR
fbLogWriter(
fbLogWriter.sFileName := '/usr/local/logs/update_log.txt';
fbLogWriter.sData := sMessage + Char(13) + Char(10);
fbLogWriter.bExecute := TRUE;
WriteLog := fbLogWriter.bDone;
END_METHOD

END_FUNCTION_BLOCK

// ---- POUs/System/PowerControl/fb_measurementCheck.TcPOU
FUNCTION_BLOCK fb_measurementCheck
VAR_IN_OUT
	r_in : REAL;
END_VAR
VAR_INPUT
	b_externalFault : BOOL;
	r_LowLimit	 	: REAL;
	r_HighLimit		: REAL;
	by_Mode			: BYTE := 0; // 0= min, 1= avg, 2= Max, 3=SUM
END_VAR

VAR
	by_InputOK		: BYTE;
END_VAR

VAR_OUTPUT
	r_Out			: REAL;
	Q				: BOOL;
END_VAR


//Check if values are within set ranges
by_InputOK.0 := r_in > r_LowLimit AND r_in < r_HighLimit;
by_InputOK.1 := r_in[Phases.L1] > r_LowLimit AND r_in[phases.L1] < r_HighLimit;
by_InputOK.2 := r_in[Phases.L2] > r_LowLimit AND r_in[phases.L2] < r_HighLimit;
by_InputOK.3 := r_in[Phases.L3] > r_LowLimit AND r_in[phases.L3] < r_HighLimit;

//Check if deviation between values is not too high

IF by_InputOK >= 14 AND NOT b_ExternalFault THEN // 14 == L1, L2, L3 OK
	CASE by_Mode OF
		0: r_out := MIN(r_in[1], r_in[2], r_in[3]); //MIN
		1: r_out := (r_in[1] + r_in[2] + r_in[3]) / 3; // AVG
		2: r_out := MAX(r_in[1], r_in[2], r_in[3]); //MAX
		3: r_out := r_in[1] + r_in[2] + r_in[3]; //sum
		4: r_out := MAX(ABS(r_in[1]), ABS(r_in[2]), ABS(r_in[3])) * 3 * SEL(r_in[1] + r_in[2] + r_in[3] < 0, 1, -1); //sum
	END_CASE
	Q := TRUE;
ELSIF by_InputOK = 1 THEN
	r_Out := r_in[0];
ELSE
	r_out := 0;
	Q := FALSE;
END_IF

END_FUNCTION_BLOCK
